LIN {X 0,Y 728.107,Z 330.531,A -85,B 0,C 180,E1 34678.19,E2 34678.19} C_VEL
LIN {X 0,Y 728.082,Z 330.529,A -85,B 0,C 180,E1 34675.632,E2 34675.632} C_VEL
LIN {X 0,Y 728.118,Z 330.525,A -85,B 0,C 180,E1 34673.04,E2 34673.04} C_VEL
LIN {X 0,Y 728.107,Z 330.532,A -85,B 0,C 180,E1 34669.995,E2 34669.995} C_VEL
LIN {X 0,Y 728.078,Z 330.53,A -85,B 0,C 180,E1 34667.503,E2 34667.503} C_VEL
LIN {X 0,Y 728.087,Z 330.528,A -85,B 0,C 180,E1 34665.043,E2 34665.043} C_VEL
LIN {X 0,Y 728.156,Z 330.532,A -85,B 0,C 180,E1 34662.12,E2 34662.12} C_VEL
LIN {X 0,Y 728.078,Z 330.532,A -85,B 0,C 180,E1 34659.406,E2 34659.406} C_VEL
LIN {X 0,Y 728.072,Z 330.53,A -85,B 0,C 180,E1 34657.021,E2 34657.021} C_VEL
LIN {X 0,Y 728.11,Z 330.528,A -85,B 0,C 180,E1 34654.44,E2 34654.44} C_VEL
LIN {X 0,Y 728.094,Z 330.533,A -85,B 0,C 180,E1 34651.416,E2 34651.416} C_VEL
LIN {X 0,Y 728.067,Z 330.532,A -85,B 0,C 180,E1 34648.977,E2 34648.977} C_VEL
LIN {X 0,Y 728.067,Z 330.527,A -85,B 0,C 180,E1 34646.615,E2 34646.615} C_VEL
LIN {X 0,Y 728.135,Z 330.531,A -85,B 0,C 180,E1 34643.93,E2 34643.93} C_VEL
LIN {X 0,Y 728.076,Z 330.534,A -85,B 0,C 180,E1 34640.993,E2 34640.993} C_VEL
LIN {X 0,Y 728.059,Z 330.532,A -85,B 0,C 180,E1 34638.594,E2 34638.594} C_VEL
LIN {X 0,Y 728.063,Z 330.531,A -85,B 0,C 180,E1 34636.256,E2 34636.256} C_VEL
LIN {X 0,Y 728.155,Z 330.51,A -85,B 0,C 180,E1 34633.433,E2 34633.433} C_VEL
LIN {X 0,Y 728.062,Z 330.521,A -85,B 0,C 180,E1 34630.589,E2 34630.589} C_VEL
LIN {X 0,Y 728.054,Z 330.543,A -85,B 0,C 180,E1 34628.235,E2 34628.235} C_VEL
LIN {X 0,Y 728.15,Z 330.769,A -85,B 0,C 180,E1 34627.473,E2 34627.473} C_VEL
LIN {X 0,Y 728.586,Z 332.326,A -85,B 0,C 180,E1 34627.328,E2 34627.328} C_VEL
LIN {X 0,Y 730.719,Z 335.448,A -85,B 0,C 180,E1 34627.132,E2 34627.132} C_VEL
LIN {X 0,Y 735.609,Z 342.898,A -85,B 0,C 180,E1 34626.692,E2 34626.692} C_VEL
LIN {X 0,Y 734.695,Z 558.029,A -85,B 0,C 180,E1 34624.049,E2 34624.049} C_VEL
LIN {X 0,Y 733.863,Z 756.602,A -85,B 0,C 180,E1 34621.662,E2 34621.662} C_VEL
LIN {X 0,Y 733.596,Z 783.313,A -85,B 0,C 180,E1 34621.191,E2 34621.191} C_VEL
LIN {X 0,Y 733.226,Z 810.458,A -85,B 0,C 180,E1 34620.549,E2 34620.549} C_VEL
LIN {X 0,Y 732.845,Z 834.995,A -85,B 0,C 180,E1 34619.817,E2 34619.817} C_VEL
LIN {X 0,Y 732.412,Z 860.75,A -85,B 0,C 180,E1 34618.903,E2 34618.903} C_VEL
LIN {X 0,Y 731.841,Z 885.617,A -85,B 0,C 180,E1 34617.854,E2 34617.854} C_VEL
LIN {X 0,Y 731.403,Z 907.627,A -85,B 0,C 180,E1 34616.789,E2 34616.789} C_VEL
LIN {X 0,Y 730.936,Z 931.895,A -85,B 0,C 180,E1 34615.458,E2 34615.458} C_VEL
LIN {X 0,Y 730.401,Z 953.79,A -85,B 0,C 180,E1 34614.085,E2 34614.085} C_VEL
LIN {X 0,Y 729.994,Z 973.19,A -85,B 0,C 180,E1 34612.732,E2 34612.732} C_VEL
LIN {X 0,Y 729.606,Z 994.463,A -85,B 0,C 180,E1 34611.077,E2 34611.077} C_VEL
LIN {X 0,Y 729.185,Z 1012.918,A -85,B 0,C 180,E1 34609.462,E2 34609.462} C_VEL
LIN {X 0,Y 728.928,Z 1030.13,A -85,B 0,C 180,E1 34607.794,E2 34607.794} C_VEL
LIN {X 0,Y 728.606,Z 1047.766,A -85,B 0,C 180,E1 34605.868,E2 34605.868} C_VEL
LIN {X 0,Y 728.411,Z 1061.269,A -85,B 0,C 180,E1 34604.214,E2 34604.214} C_VEL
LIN {X 0,Y 728.279,Z 1073.883,A -85,B 0,C 180,E1 34602.493,E2 34602.493} C_VEL
LIN {X 0,Y 728.122,Z 1087.68,A -85,B 0,C 180,E1 34600.347,E2 34600.347} C_VEL
LIN {X 0,Y 728.035,Z 1097.981,A -85,B 0,C 180,E1 34598.474,E2 34598.474} C_VEL
LIN {X 0,Y 727.947,Z 1105.598,A -85,B 0,C 180,E1 34596.888,E2 34596.888} C_VEL
LIN {X 0,Y 727.935,Z 1112.65,A -85,B 0,C 180,E1 34595.187,E2 34595.187} C_VEL
LIN {X 0,Y 727.924,Z 1118.773,A -85,B 0,C 180,E1 34593.424,E2 34593.424} C_VEL
LIN {X 0,Y 727.924,Z 1124.47,A -85,B 0,C 180,E1 34591.373,E2 34591.373} C_VEL
LIN {X 0,Y 727.915,Z 1128.569,A -85,B 0,C 180,E1 34589.276,E2 34589.276} C_VEL
LIN {X 0,Y 727.873,Z 1130.818,A -85,B 0,C 180,E1 34587.4,E2 34587.4} C_VEL
LIN {X 0,Y 727.906,Z 1131.802,A -85,B 0,C 180,E1 34585.697,E2 34585.697} C_VEL
LIN {X 0,Y 727.896,Z 1131.74,A -85,B 0,C 180,E1 34583.992,E2 34583.992} C_VEL
LIN {X 0,Y 727.916,Z 1130.33,A -85,B 0,C 180,E1 34581.94,E2 34581.94} C_VEL
LIN {X 0,Y 727.92,Z 1127.194,A -85,B 0,C 180,E1 34579.834,E2 34579.834} C_VEL
LIN {X 0,Y 727.93,Z 1122.518,A -85,B 0,C 180,E1 34577.755,E2 34577.755} C_VEL
LIN {X 0,Y 727.952,Z 1115.426,A -85,B 0,C 180,E1 34575.455,E2 34575.455} C_VEL
LIN {X 0,Y 727.985,Z 1107.016,A -85,B 0,C 180,E1 34573.341,E2 34573.341} C_VEL
LIN {X 0,Y 728.024,Z 1099.06,A -85,B 0,C 180,E1 34571.648,E2 34571.648} C_VEL
LIN {X 0,Y 728.063,Z 1089.98,A -85,B 0,C 180,E1 34569.965,E2 34569.965} C_VEL
LIN {X 0,Y 728.178,Z 1080.234,A -85,B 0,C 180,E1 34568.369,E2 34568.369} C_VEL
LIN {X 0,Y 728.35,Z 1067.162,A -85,B 0,C 180,E1 34566.464,E2 34566.464} C_VEL
LIN {X 0,Y 728.57,Z 1051.53,A -85,B 0,C 180,E1 34564.487,E2 34564.487} C_VEL
LIN {X 0,Y 728.777,Z 1037.612,A -85,B 0,C 180,E1 34562.91,E2 34562.91} C_VEL
LIN {X 0,Y 729.073,Z 1021.129,A -85,B 0,C 180,E1 34561.218,E2 34561.218} C_VEL
LIN {X 0,Y 729.412,Z 1001.74,A -85,B 0,C 180,E1 34559.45,E2 34559.45} C_VEL
LIN {X 0,Y 729.794,Z 983.502,A -85,B 0,C 180,E1 34557.959,E2 34557.959} C_VEL
LIN {X 0,Y 730.292,Z 961.036,A -85,B 0,C 180,E1 34556.31,E2 34556.31} C_VEL
LIN {X 0,Y 730.693,Z 939.861,A -85,B 0,C 180,E1 34554.936,E2 34554.936} C_VEL
LIN {X 0,Y 731.173,Z 918.904,A -85,B 0,C 180,E1 34553.719,E2 34553.719} C_VEL
LIN {X 0,Y 731.75,Z 892.704,A -85,B 0,C 180,E1 34552.383,E2 34552.383} C_VEL
LIN {X 0,Y 732.175,Z 869.485,A -85,B 0,C 180,E1 34551.36,E2 34551.36} C_VEL
LIN {X 0,Y 732.587,Z 846.861,A -85,B 0,C 180,E1 34550.494,E2 34550.494} C_VEL
LIN {X 0,Y 733.091,Z 818.282,A -85,B 0,C 180,E1 34549.578,E2 34549.578} C_VEL
LIN {X 0,Y 733.499,Z 791.667,A -85,B 0,C 180,E1 34548.898,E2 34548.898} C_VEL
LIN {X 0,Y 733.775,Z 764.714,A -85,B 0,C 180,E1 34548.375,E2 34548.375} C_VEL
LIN {X 0,Y 734.007,Z 735.424,A -85,B 0,C 180,E1 34547.977,E2 34547.977} C_VEL
LIN {X 0,Y 734.916,Z 505.975,A -85,B 0,C 180,E1 34545.23,E2 34545.23} C_VEL
LIN {X 0,Y 735.52,Z 342.703,A -85,B 0,C 180,E1 34543.209,E2 34543.209} C_VEL
LIN {X 0,Y 731.351,Z 336.17,A -85,B 0,C 180,E1 34542.832,E2 34542.832} C_VEL
LIN {X 0,Y 728.754,Z 332.691,A -85,B 0,C 180,E1 34542.601,E2 34542.601} C_VEL
LIN {X 0,Y 728.209,Z 330.851,A -85,B 0,C 180,E1 34542.459,E2 34542.459} C_VEL
LIN {X 0,Y 728.09,Z 330.538,A -85,B 0,C 180,E1 34541.753,E2 34541.753} C_VEL
LIN {X 0,Y 728.105,Z 330.514,A -85,B 0,C 180,E1 34539.165,E2 34539.165} C_VEL
LIN {X 0,Y 728.155,Z 330.527,A -85,B 0,C 180,E1 34536.189,E2 34536.189} C_VEL
LIN {X 0,Y 728.106,Z 330.53,A -85,B 0,C 180,E1 34533.379,E2 34533.379} C_VEL
LIN {X 0,Y 728.158,Z 330.533,A -85,B 0,C 180,E1 34530.554,E2 34530.554} C_VEL
LIN {X 0,Y 728.13,Z 330.526,A -85,B 0,C 180,E1 34527.618,E2 34527.618} C_VEL
LIN {X 0,Y 728.144,Z 330.534,A -85,B 0,C 180,E1 34524.778,E2 34524.778} C_VEL
LIN {X 0,Y 728.156,Z 330.527,A -85,B 0,C 180,E1 34521.734,E2 34521.734} C_VEL
LIN {X 0,Y 728.161,Z 330.717,A -85,B 0,C 180,E1 34519.286,E2 34519.286} C_VEL
LIN {X 0,Y 729.649,Z 334.269,A -85,B 0,C 180,E1 34518.869,E2 34518.869} C_VEL
LIN {X 0,Y 730.762,Z 336.329,A -85,B 0,C 180,E1 34518.633,E2 34518.633} C_VEL
LIN {X 0,Y 735.297,Z 345.332,A -85,B 0,C 180,E1 34517.648,E2 34517.648} C_VEL
LIN {X 0,Y 734.588,Z 386.425,A -85,B 0,C 180,E1 34515.111,E2 34515.111} C_VEL
LIN {X 0,Y 734.124,Z 427.552,A -85,B 0,C 180,E1 34512.689,E2 34512.689} C_VEL
LIN {X 0,Y 735.825,Z 435.852,A -85,B 0,C 180,E1 34512.457,E2 34512.457} C_VEL
LIN {X 0,Y 734.955,Z 645.516,A -85,B 0,C 180,E1 34509.852,E2 34509.852} C_VEL
LIN {X 0,Y 734.064,Z 871.192,A -85,B 0,C 180,E1 34507.146,E2 34507.146} C_VEL
LIN {X 0,Y 733.843,Z 910.622,A -85,B 0,C 180,E1 34506.646,E2 34506.646} C_VEL
LIN {X 0,Y 733.519,Z 937.557,A -85,B 0,C 180,E1 34506.146,E2 34506.146} C_VEL
LIN {X 0,Y 733.177,Z 963.48,A -85,B 0,C 180,E1 34505.511,E2 34505.511} C_VEL
LIN {X 0,Y 732.755,Z 991.376,A -85,B 0,C 180,E1 34504.654,E2 34504.654} C_VEL
LIN {X 0,Y 732.218,Z 1016.477,A -85,B 0,C 180,E1 34503.717,E2 34503.717} C_VEL
LIN {X 0,Y 731.801,Z 1037.586,A -85,B 0,C 180,E1 34502.807,E2 34502.807} C_VEL
LIN {X 0,Y 731.382,Z 1059.085,A -85,B 0,C 180,E1 34501.758,E2 34501.758} C_VEL
LIN {X 0,Y 730.853,Z 1084.154,A -85,B 0,C 180,E1 34500.365,E2 34500.365} C_VEL
LIN {X 0,Y 730.378,Z 1104.565,A -85,B 0,C 180,E1 34499.077,E2 34499.077} C_VEL
LIN {X 0,Y 730.013,Z 1122.255,A -85,B 0,C 180,E1 34497.843,E2 34497.843} C_VEL
LIN {X 0,Y 729.634,Z 1143.199,A -85,B 0,C 180,E1 34496.228,E2 34496.228} C_VEL
LIN {X 0,Y 729.209,Z 1161.707,A -85,B 0,C 180,E1 34494.617,E2 34494.617} C_VEL
LIN {X 0,Y 728.956,Z 1177.537,A -85,B 0,C 180,E1 34493.097,E2 34493.097} C_VEL
LIN {X 0,Y 728.684,Z 1194.989,A -85,B 0,C 180,E1 34491.238,E2 34491.238} C_VEL
LIN {X 0,Y 728.438,Z 1210.158,A -85,B 0,C 180,E1 34489.401,E2 34489.401} C_VEL
LIN {X 0,Y 728.264,Z 1221.836,A -85,B 0,C 180,E1 34487.828,E2 34487.828} C_VEL
LIN {X 0,Y 728.149,Z 1232.784,A -85,B 0,C 180,E1 34486.186,E2 34486.186} C_VEL
LIN {X 0,Y 728.086,Z 1244.308,A -85,B 0,C 180,E1 34484.23,E2 34484.23} C_VEL
LIN {X 0,Y 727.973,Z 1254.716,A -85,B 0,C 180,E1 34482.131,E2 34482.131} C_VEL
LIN {X 0,Y 727.956,Z 1261.878,A -85,B 0,C 180,E1 34480.431,E2 34480.431} C_VEL
LIN {X 0,Y 727.916,Z 1267.792,A -85,B 0,C 180,E1 34478.77,E2 34478.77} C_VEL
LIN {X 0,Y 727.917,Z 1273.175,A -85,B 0,C 180,E1 34476.943,E2 34476.943} C_VEL
LIN {X 0,Y 727.911,Z 1277.782,A -85,B 0,C 180,E1 34474.806,E2 34474.806} C_VEL
LIN {X 0,Y 727.912,Z 1280.541,A -85,B 0,C 180,E1 34472.756,E2 34472.756} C_VEL
LIN {X 0,Y 727.874,Z 1281.715,A -85,B 0,C 180,E1 34471.023,E2 34471.023} C_VEL
LIN {X 0,Y 727.863,Z 1281.827,A -85,B 0,C 180,E1 34469.37,E2 34469.37} C_VEL
LIN {X 0,Y 727.907,Z 1280.946,A -85,B 0,C 180,E1 34467.717,E2 34467.717} C_VEL
LIN {X 0,Y 727.919,Z 1278.803,A -85,B 0,C 180,E1 34465.825,E2 34465.825} C_VEL
LIN {X 0,Y 727.925,Z 1274.734,A -85,B 0,C 180,E1 34463.691,E2 34463.691} C_VEL
LIN {X 0,Y 727.939,Z 1269.073,A -85,B 0,C 180,E1 34461.628,E2 34461.628} C_VEL
LIN {X 0,Y 727.956,Z 1263.045,A -85,B 0,C 180,E1 34459.874,E2 34459.874} C_VEL
LIN {X 0,Y 727.966,Z 1256.145,A -85,B 0,C 180,E1 34458.191,E2 34458.191} C_VEL
LIN {X 0,Y 727.993,Z 1248.883,A -85,B 0,C 180,E1 34456.659,E2 34456.659} C_VEL
LIN {X 0,Y 728.086,Z 1240.595,A -85,B 0,C 180,E1 34455.119,E2 34455.119} C_VEL
LIN {X 0,Y 728.177,Z 1230.694,A -85,B 0,C 180,E1 34453.487,E2 34453.487} C_VEL
LIN {X 0,Y 728.347,Z 1218.342,A -85,B 0,C 180,E1 34451.677,E2 34451.677} C_VEL
LIN {X 0,Y 728.544,Z 1202.255,A -85,B 0,C 180,E1 34449.617,E2 34449.617} C_VEL
LIN {X 0,Y 728.752,Z 1188.057,A -85,B 0,C 180,E1 34448.002,E2 34448.002} C_VEL
LIN {X 0,Y 729.047,Z 1172.216,A -85,B 0,C 180,E1 34446.372,E2 34446.372} C_VEL
LIN {X 0,Y 729.421,Z 1152.324,A -85,B 0,C 180,E1 34444.548,E2 34444.548} C_VEL
LIN {X 0,Y 729.734,Z 1134.945,A -85,B 0,C 180,E1 34443.117,E2 34443.117} C_VEL
LIN {X 0,Y 730.18,Z 1115.658,A -85,B 0,C 180,E1 34441.679,E2 34441.679} C_VEL
LIN {X 0,Y 730.668,Z 1092.159,A -85,B 0,C 180,E1 34440.125,E2 34440.125} C_VEL
LIN {X 0,Y 731.057,Z 1072.423,A -85,B 0,C 180,E1 34438.961,E2 34438.961} C_VEL
LIN {X 0,Y 731.515,Z 1051.962,A -85,B 0,C 180,E1 34437.879,E2 34437.879} C_VEL
LIN {X 0,Y 732.098,Z 1026.541,A -85,B 0,C 180,E1 34436.699,E2 34436.699} C_VEL
LIN {X 0,Y 732.503,Z 1003.39,A -85,B 0,C 180,E1 34435.779,E2 34435.779} C_VEL
LIN {X 0,Y 732.865,Z 981.835,A -85,B 0,C 180,E1 34435.039,E2 34435.039} C_VEL
LIN {X 0,Y 733.236,Z 959.117,A -85,B 0,C 180,E1 34434.371,E2 34434.371} C_VEL
LIN {X 0,Y 733.615,Z 932.145,A -85,B 0,C 180,E1 34433.739,E2 34433.739} C_VEL
LIN {X 0,Y 733.88,Z 904.403,A -85,B 0,C 180,E1 34433.261,E2 34433.261} C_VEL
LIN {X 0,Y 734.857,Z 667.496,A -85,B 0,C 180,E1 34430.415,E2 34430.415} C_VEL
LIN {X 0,Y 735.696,Z 465.373,A -85,B 0,C 180,E1 34427.915,E2 34427.915} C_VEL
LIN {X 0,Y 735.645,Z 434.163,A -85,B 0,C 180,E1 34427.508,E2 34427.508} C_VEL
LIN {X 0,Y 734.005,Z 426.794,A -85,B 0,C 180,E1 34427.282,E2 34427.282} C_VEL
LIN {X 0,Y 734.649,Z 382.935,A -85,B 0,C 180,E1 34424.678,E2 34424.678} C_VEL
LIN {X 0,Y 735.253,Z 345.215,A -85,B 0,C 180,E1 34422.341,E2 34422.341} C_VEL
LIN {X 0,Y 731.832,Z 338.52,A -85,B 0,C 180,E1 34421.607,E2 34421.607} C_VEL
LIN {X 0,Y 730.082,Z 334.806,A -85,B 0,C 180,E1 34421.205,E2 34421.205} C_VEL
LIN {X 0,Y 728.288,Z 331.373,A -85,B 0,C 180,E1 34420.807,E2 34420.807} C_VEL
LIN {X 0,Y 728.146,Z 330.583,A -85,B 0,C 180,E1 34420.661,E2 34420.661} C_VEL
LIN {X 0,Y 728.135,Z 330.495,A -85,B 0,C 180,E1 34417.768,E2 34417.768} C_VEL
LIN {X 0,Y 728.138,Z 330.533,A -85,B 0,C 180,E1 34414.934,E2 34414.934} C_VEL
LIN {X 0,Y 728.155,Z 330.523,A -85,B 0,C 180,E1 34412.009,E2 34412.009} C_VEL
LIN {X 0,Y 728.154,Z 330.53,A -85,B 0,C 180,E1 34408.99,E2 34408.99} C_VEL
LIN {X 0,Y 728.15,Z 330.52,A -85,B 0,C 180,E1 34405.98,E2 34405.98} C_VEL
LIN {X 0,Y 728.159,Z 330.532,A -85,B 0,C 180,E1 34402.868,E2 34402.868} C_VEL
LIN {X 0,Y 728.138,Z 330.523,A -85,B 0,C 180,E1 34399.911,E2 34399.911} C_VEL
LIN {X 0,Y 728.15,Z 330.529,A -85,B 0,C 180,E1 34396.925,E2 34396.925} C_VEL
LIN {X 0,Y 728.122,Z 330.527,A -85,B 0,C 180,E1 34394.068,E2 34394.068} C_VEL
LIN {X 0,Y 728.154,Z 330.52,A -85,B 0,C 180,E1 34391.244,E2 34391.244} C_VEL
LIN {X 0,Y 728.139,Z 330.531,A -85,B 0,C 180,E1 34388.29,E2 34388.29} C_VEL
LIN {X 0,Y 728.141,Z 330.52,A -85,B 0,C 180,E1 34385.358,E2 34385.358} C_VEL
LIN {X 0,Y 728.153,Z 330.53,A -85,B 0,C 180,E1 34382.282,E2 34382.282} C_VEL
LIN {X 0,Y 728.119,Z 330.525,A -85,B 0,C 180,E1 34379.449,E2 34379.449} C_VEL
LIN {X 0,Y 728.151,Z 330.525,A -85,B 0,C 180,E1 34376.615,E2 34376.615} C_VEL
LIN {X 0,Y 728.12,Z 330.529,A -85,B 0,C 180,E1 34373.693,E2 34373.693} C_VEL
LIN {X 0,Y 728.14,Z 330.522,A -85,B 0,C 180,E1 34370.867,E2 34370.867} C_VEL
LIN {X 0,Y 728.142,Z 330.532,A -85,B 0,C 180,E1 34367.791,E2 34367.791} C_VEL
LIN {X 0,Y 728.156,Z 330.524,A -85,B 0,C 180,E1 34366.385,E2 34366.385} C_VEL
LIN {X 0,Y 727.165,Z 330.656,A -85,B 0,C 180,E1 34365.779,E2 34365.779} C_VEL
LIN {X 0,Y 720.764,Z 331.456,A -85,B 0,C 180,E1 34364.081,E2 34364.081} C_VEL
LIN {X 0,Y 720.198,Z 331.519,A -85,B 0,C 180,E1 34363.64,E2 34363.64} C_VEL
LIN {X 0,Y 720.172,Z 331.515,A -85,B 0,C 180,E1 34360.873,E2 34360.873} C_VEL
LIN {X 0,Y 720.217,Z 331.516,A -85,B 0,C 180,E1 34357.985,E2 34357.985} C_VEL
LIN {X 0,Y 720.173,Z 331.519,A -85,B 0,C 180,E1 34355.122,E2 34355.122} C_VEL
LIN {X 0,Y 720.188,Z 331.513,A -85,B 0,C 180,E1 34352.346,E2 34352.346} C_VEL
LIN {X 0,Y 720.198,Z 331.521,A -85,B 0,C 180,E1 34349.247,E2 34349.247} C_VEL
LIN {X 0,Y 720.162,Z 331.516,A -85,B 0,C 180,E1 34346.55,E2 34346.55} C_VEL
LIN {X 0,Y 720.219,Z 331.511,A -85,B 0,C 180,E1 34343.742,E2 34343.742} C_VEL
LIN {X 0,Y 720.171,Z 331.519,A -85,B 0,C 180,E1 34340.78,E2 34340.78} C_VEL
LIN {X 0,Y 720.16,Z 331.515,A -85,B 0,C 180,E1 34338.206,E2 34338.206} C_VEL
LIN {X 0,Y 720.221,Z 331.517,A -85,B 0,C 180,E1 34335.3,E2 34335.3} C_VEL
LIN {X 0,Y 720.161,Z 331.518,A -85,B 0,C 180,E1 34332.436,E2 34332.436} C_VEL
LIN {X 0,Y 720.161,Z 331.516,A -85,B 0,C 180,E1 34329.843,E2 34329.843} C_VEL
LIN {X 0,Y 720.223,Z 331.519,A -85,B 0,C 180,E1 34326.951,E2 34326.951} C_VEL
LIN {X 0,Y 720.153,Z 331.519,A -85,B 0,C 180,E1 34324.12,E2 34324.12} C_VEL
LIN {X 0,Y 720.158,Z 331.516,A -85,B 0,C 180,E1 34321.563,E2 34321.563} C_VEL
LIN {X 0,Y 720.221,Z 331.519,A -85,B 0,C 180,E1 34318.617,E2 34318.617} C_VEL
LIN {X 0,Y 720.147,Z 331.519,A -85,B 0,C 180,E1 34315.847,E2 34315.847} C_VEL
LIN {X 0,Y 720.153,Z 331.515,A -85,B 0,C 180,E1 34313.31,E2 34313.31} C_VEL
LIN {X 0,Y 720.22,Z 331.519,A -85,B 0,C 180,E1 34310.393,E2 34310.393} C_VEL
LIN {X 0,Y 720.143,Z 331.519,A -85,B 0,C 180,E1 34307.619,E2 34307.619} C_VEL
LIN {X 0,Y 720.143,Z 331.517,A -85,B 0,C 180,E1 34305.131,E2 34305.131} C_VEL
LIN {X 0,Y 720.223,Z 331.519,A -85,B 0,C 180,E1 34302.263,E2 34302.263} C_VEL
LIN {X 0,Y 720.14,Z 331.521,A -85,B 0,C 180,E1 34299.43,E2 34299.43} C_VEL
LIN {X 0,Y 720.134,Z 331.519,A -85,B 0,C 180,E1 34297.018,E2 34297.018} C_VEL
LIN {X 0,Y 720.168,Z 331.517,A -85,B 0,C 180,E1 34294.459,E2 34294.459} C_VEL
LIN {X 0,Y 720.157,Z 331.522,A -85,B 0,C 180,E1 34291.432,E2 34291.432} C_VEL
LIN {X 0,Y 720.128,Z 331.521,A -85,B 0,C 180,E1 34288.966,E2 34288.966} C_VEL
LIN {X 0,Y 720.131,Z 331.515,A -85,B 0,C 180,E1 34286.577,E2 34286.577} C_VEL
LIN {X 0,Y 720.219,Z 331.516,A -85,B 0,C 180,E1 34283.74,E2 34283.74} C_VEL
LIN {X 0,Y 720.131,Z 331.523,A -85,B 0,C 180,E1 34280.893,E2 34280.893} C_VEL
LIN {X 0,Y 720.121,Z 331.521,A -85,B 0,C 180,E1 34278.548,E2 34278.548} C_VEL
LIN {X 0,Y 720.128,Z 331.52,A -85,B 0,C 180,E1 34276.183,E2 34276.183} C_VEL
LIN {X 0,Y 720.207,Z 331.5,A -85,B 0,C 180,E1 34273.299,E2 34273.299} C_VEL
LIN {X 0,Y 720.12,Z 331.508,A -85,B 0,C 180,E1 34270.527,E2 34270.527} C_VEL
LIN {X 0,Y 720.115,Z 331.532,A -85,B 0,C 180,E1 34268.24,E2 34268.24} C_VEL
LIN {X 0,Y 720.148,Z 331.744,A -85,B 0,C 180,E1 34268.047,E2 34268.047} C_VEL
LIN {X 0,Y 720.558,Z 333.301,A -85,B 0,C 180,E1 34267.9,E2 34267.9} C_VEL
LIN {X 0,Y 722.666,Z 336.411,A -85,B 0,C 180,E1 34267.7,E2 34267.7} C_VEL
LIN {X 0,Y 723.885,Z 338.005,A -85,B 0,C 180,E1 34267.59,E2 34267.59} C_VEL
LIN {X 0,Y 729.608,Z 346.693,A -85,B 0,C 180,E1 34267.065,E2 34267.065} C_VEL
LIN {X 0,Y 728.452,Z 562.734,A -85,B 0,C 180,E1 34264.39,E2 34264.39} C_VEL
LIN {X 0,Y 727.429,Z 756.797,A -85,B 0,C 180,E1 34262.038,E2 34262.038} C_VEL
LIN {X 0,Y 727.091,Z 783.495,A -85,B 0,C 180,E1 34261.563,E2 34261.563} C_VEL
LIN {X 0,Y 726.621,Z 810.696,A -85,B 0,C 180,E1 34260.915,E2 34260.915} C_VEL
LIN {X 0,Y 726.143,Z 835.479,A -85,B 0,C 180,E1 34260.17,E2 34260.17} C_VEL
LIN {X 0,Y 725.597,Z 861.061,A -85,B 0,C 180,E1 34259.254,E2 34259.254} C_VEL
LIN {X 0,Y 724.916,Z 885.709,A -85,B 0,C 180,E1 34258.204,E2 34258.204} C_VEL
LIN {X 0,Y 724.343,Z 907.446,A -85,B 0,C 180,E1 34257.147,E2 34257.147} C_VEL
LIN {X 0,Y 723.75,Z 932.011,A -85,B 0,C 180,E1 34255.787,E2 34255.787} C_VEL
LIN {X 0,Y 723.094,Z 953.932,A -85,B 0,C 180,E1 34254.398,E2 34254.398} C_VEL
LIN {X 0,Y 722.552,Z 973.986,A -85,B 0,C 180,E1 34252.985,E2 34252.985} C_VEL
LIN {X 0,Y 722.007,Z 996.432,A -85,B 0,C 180,E1 34251.202,E2 34251.202} C_VEL
LIN {X 0,Y 721.525,Z 1014.133,A -85,B 0,C 180,E1 34249.625,E2 34249.625} C_VEL
LIN {X 0,Y 721.172,Z 1032.083,A -85,B 0,C 180,E1 34247.852,E2 34247.852} C_VEL
LIN {X 0,Y 720.786,Z 1048.868,A -85,B 0,C 180,E1 34245.974,E2 34245.974} C_VEL
LIN {X 0,Y 720.55,Z 1062.067,A -85,B 0,C 180,E1 34244.328,E2 34244.328} C_VEL
LIN {X 0,Y 720.359,Z 1075.904,A -85,B 0,C 180,E1 34242.402,E2 34242.402} C_VEL
LIN {X 0,Y 720.154,Z 1088.984,A -85,B 0,C 180,E1 34240.291,E2 34240.291} C_VEL
LIN {X 0,Y 720.068,Z 1098.26,A -85,B 0,C 180,E1 34238.571,E2 34238.571} C_VEL
LIN {X 0,Y 719.967,Z 1106.244,A -85,B 0,C 180,E1 34236.876,E2 34236.876} C_VEL
LIN {X 0,Y 719.946,Z 1113.054,A -85,B 0,C 180,E1 34235.196,E2 34235.196} C_VEL
LIN {X 0,Y 719.922,Z 1119.257,A -85,B 0,C 180,E1 34233.367,E2 34233.367} C_VEL
LIN {X 0,Y 719.922,Z 1124.818,A -85,B 0,C 180,E1 34231.295,E2 34231.295} C_VEL
LIN {X 0,Y 719.912,Z 1128.941,A -85,B 0,C 180,E1 34229.086,E2 34229.086} C_VEL
LIN {X 0,Y 719.863,Z 1131.019,A -85,B 0,C 180,E1 34227.193,E2 34227.193} C_VEL
LIN {X 0,Y 719.898,Z 1131.885,A -85,B 0,C 180,E1 34225.416,E2 34225.416} C_VEL
LIN {X 0,Y 719.88,Z 1131.454,A -85,B 0,C 180,E1 34223.233,E2 34223.233} C_VEL
LIN {X 0,Y 719.907,Z 1129.265,A -85,B 0,C 180,E1 34221.039,E2 34221.039} C_VEL
LIN {X 0,Y 719.911,Z 1125.392,A -85,B 0,C 180,E1 34218.882,E2 34218.882} C_VEL
LIN {X 0,Y 719.905,Z 1120.297,A -85,B 0,C 180,E1 34216.873,E2 34216.873} C_VEL
LIN {X 0,Y 719.956,Z 1113.563,A -85,B 0,C 180,E1 34214.849,E2 34214.849} C_VEL
LIN {X 0,Y 719.985,Z 1106.46,A -85,B 0,C 180,E1 34213.083,E2 34213.083} C_VEL
LIN {X 0,Y 720.07,Z 1098.432,A -85,B 0,C 180,E1 34211.372,E2 34211.372} C_VEL
LIN {X 0,Y 720.159,Z 1088.824,A -85,B 0,C 180,E1 34209.591,E2 34209.591} C_VEL
LIN {X 0,Y 720.344,Z 1075.833,A -85,B 0,C 180,E1 34207.497,E2 34207.497} C_VEL
LIN {X 0,Y 720.553,Z 1062.015,A -85,B 0,C 180,E1 34205.574,E2 34205.574} C_VEL
LIN {X 0,Y 720.792,Z 1048.542,A -85,B 0,C 180,E1 34203.898,E2 34203.898} C_VEL
LIN {X 0,Y 721.189,Z 1031.4,A -85,B 0,C 180,E1 34201.986,E2 34201.986} C_VEL
LIN {X 0,Y 721.557,Z 1013.64,A -85,B 0,C 180,E1 34200.238,E2 34200.238} C_VEL
LIN {X 0,Y 722.059,Z 994.848,A -85,B 0,C 180,E1 34198.572,E2 34198.572} C_VEL
LIN {X 0,Y 722.564,Z 973.172,A -85,B 0,C 180,E1 34196.867,E2 34196.867} C_VEL
LIN {X 0,Y 723.091,Z 954.05,A -85,B 0,C 180,E1 34195.519,E2 34195.519} C_VEL
LIN {X 0,Y 723.776,Z 930.803,A -85,B 0,C 180,E1 34194.053,E2 34194.053} C_VEL
LIN {X 0,Y 724.345,Z 907.034,A -85,B 0,C 180,E1 34192.744,E2 34192.744} C_VEL
LIN {X 0,Y 724.909,Z 885.87,A -85,B 0,C 180,E1 34191.712,E2 34191.712} C_VEL
LIN {X 0,Y 725.571,Z 861.66,A -85,B 0,C 180,E1 34190.681,E2 34190.681} C_VEL
LIN {X 0,Y 726.123,Z 836.305,A -85,B 0,C 180,E1 34189.768,E2 34189.768} C_VEL
LIN {X 0,Y 726.608,Z 811.727,A -85,B 0,C 180,E1 34189.023,E2 34189.023} C_VEL
LIN {X 0,Y 727.064,Z 784.919,A -85,B 0,C 180,E1 34188.377,E2 34188.377} C_VEL
LIN {X 0,Y 727.414,Z 758.626,A -85,B 0,C 180,E1 34187.9,E2 34187.9} C_VEL
LIN {X 0,Y 727.769,Z 701.915,A -85,B 0,C 180,E1 34187.198,E2 34187.198} C_VEL
LIN {X 0,Y 728.907,Z 476.652,A -85,B 0,C 180,E1 34184.466,E2 34184.466} C_VEL
LIN {X 0,Y 729.437,Z 346.129,A -85,B 0,C 180,E1 34182.826,E2 34182.826} C_VEL
LIN {X 0,Y 723.601,Z 337.376,A -85,B 0,C 180,E1 34182.291,E2 34182.291} C_VEL
LIN {X 0,Y 720.89,Z 333.973,A -85,B 0,C 180,E1 34182.047,E2 34182.047} C_VEL
LIN {X 0,Y 720.251,Z 332.085,A -85,B 0,C 180,E1 34181.924,E2 34181.924} C_VEL
LIN {X 0,Y 720.154,Z 331.54,A -85,B 0,C 180,E1 34181.746,E2 34181.746} C_VEL
LIN {X 0,Y 720.169,Z 331.501,A -85,B 0,C 180,E1 34179.129,E2 34179.129} C_VEL
LIN {X 0,Y 720.205,Z 331.517,A -85,B 0,C 180,E1 34176.084,E2 34176.084} C_VEL
LIN {X 0,Y 720.167,Z 331.52,A -85,B 0,C 180,E1 34173.355,E2 34173.355} C_VEL
LIN {X 0,Y 720.219,Z 331.521,A -85,B 0,C 180,E1 34170.512,E2 34170.512} C_VEL
LIN {X 0,Y 720.189,Z 331.516,A -85,B 0,C 180,E1 34167.577,E2 34167.577} C_VEL
LIN {X 0,Y 720.211,Z 331.523,A -85,B 0,C 180,E1 34164.719,E2 34164.719} C_VEL
LIN {X 0,Y 720.214,Z 331.518,A -85,B 0,C 180,E1 34161.641,E2 34161.641} C_VEL
LIN {X 0,Y 720.235,Z 331.731,A -85,B 0,C 180,E1 34159.956,E2 34159.956} C_VEL
LIN {X 0,Y 721.517,Z 334.966,A -85,B 0,C 180,E1 34159.566,E2 34159.566} C_VEL
LIN {X 0,Y 722.775,Z 337.218,A -85,B 0,C 180,E1 34159.296,E2 34159.296} C_VEL
LIN {X 0,Y 729.17,Z 349.743,A -85,B 0,C 180,E1 34157.889,E2 34157.889} C_VEL
LIN {X 0,Y 728.284,Z 390.899,A -85,B 0,C 180,E1 34155.33,E2 34155.33} C_VEL
LIN {X 0,Y 727.609,Z 426.819,A -85,B 0,C 180,E1 34153.184,E2 34153.184} C_VEL
LIN {X 0,Y 729.898,Z 437.785,A -85,B 0,C 180,E1 34152.859,E2 34152.859} C_VEL
LIN {X 0,Y 728.796,Z 647.017,A -85,B 0,C 180,E1 34150.239,E2 34150.239} C_VEL
LIN {X 0,Y 727.672,Z 872.536,A -85,B 0,C 180,E1 34147.511,E2 34147.511} C_VEL
LIN {X 0,Y 727.398,Z 911.215,A -85,B 0,C 180,E1 34147.015,E2 34147.015} C_VEL
LIN {X 0,Y 726.991,Z 938.374,A -85,B 0,C 180,E1 34146.504,E2 34146.504} C_VEL
LIN {X 0,Y 726.56,Z 964.191,A -85,B 0,C 180,E1 34145.864,E2 34145.864} C_VEL
LIN {X 0,Y 726.021,Z 991.909,A -85,B 0,C 180,E1 34145.002,E2 34145.002} C_VEL
LIN {X 0,Y 725.376,Z 1016.909,A -85,B 0,C 180,E1 34144.06,E2 34144.06} C_VEL
LIN {X 0,Y 724.836,Z 1038.081,A -85,B 0,C 180,E1 34143.139,E2 34143.139} C_VEL
LIN {X 0,Y 724.294,Z 1060.252,A -85,B 0,C 180,E1 34142.045,E2 34142.045} C_VEL
LIN {X 0,Y 723.607,Z 1085.615,A -85,B 0,C 180,E1 34140.61,E2 34140.61} C_VEL
LIN {X 0,Y 723.048,Z 1105.229,A -85,B 0,C 180,E1 34139.355,E2 34139.355} C_VEL
LIN {X 0,Y 722.551,Z 1124.265,A -85,B 0,C 180,E1 34138.007,E2 34138.007} C_VEL
LIN {X 0,Y 721.989,Z 1146.754,A -85,B 0,C 180,E1 34136.217,E2 34136.217} C_VEL
LIN {X 0,Y 721.54,Z 1163.38,A -85,B 0,C 180,E1 34134.74,E2 34134.74} C_VEL
LIN {X 0,Y 721.209,Z 1180.093,A -85,B 0,C 180,E1 34133.101,E2 34133.101} C_VEL
LIN {X 0,Y 720.833,Z 1197.834,A -85,B 0,C 180,E1 34131.14,E2 34131.14} C_VEL
LIN {X 0,Y 720.568,Z 1211.449,A -85,B 0,C 180,E1 34129.453,E2 34129.453} C_VEL
LIN {X 0,Y 720.35,Z 1223.584,A -85,B 0,C 180,E1 34127.78,E2 34127.78} C_VEL
LIN {X 0,Y 720.209,Z 1236.873,A -85,B 0,C 180,E1 34125.707,E2 34125.707} C_VEL
LIN {X 0,Y 720.048,Z 1247.243,A -85,B 0,C 180,E1 34123.818,E2 34123.818} C_VEL
LIN {X 0,Y 719.992,Z 1255.336,A -85,B 0,C 180,E1 34122.126,E2 34122.126} C_VEL
LIN {X 0,Y 719.964,Z 1262.128,A -85,B 0,C 180,E1 34120.482,E2 34120.482} C_VEL
LIN {X 0,Y 719.92,Z 1268.049,A -85,B 0,C 180,E1 34118.788,E2 34118.788} C_VEL
LIN {X 0,Y 719.919,Z 1273.37,A -85,B 0,C 180,E1 34116.94,E2 34116.94} C_VEL
LIN {X 0,Y 719.91,Z 1277.928,A -85,B 0,C 180,E1 34114.78,E2 34114.78} C_VEL
LIN {X 0,Y 719.91,Z 1280.609,A -85,B 0,C 180,E1 34112.707,E2 34112.707} C_VEL
LIN {X 0,Y 719.869,Z 1281.737,A -85,B 0,C 180,E1 34110.955,E2 34110.955} C_VEL
LIN {X 0,Y 719.863,Z 1281.827,A -85,B 0,C 180,E1 34109.363,E2 34109.363} C_VEL
LIN {X 0,Y 719.906,Z 1280.946,A -85,B 0,C 180,E1 34107.692,E2 34107.692} C_VEL
LIN {X 0,Y 719.92,Z 1278.803,A -85,B 0,C 180,E1 34105.779,E2 34105.779} C_VEL
LIN {X 0,Y 719.927,Z 1274.734,A -85,B 0,C 180,E1 34103.621,E2 34103.621} C_VEL
LIN {X 0,Y 719.944,Z 1269.073,A -85,B 0,C 180,E1 34101.534,E2 34101.534} C_VEL
LIN {X 0,Y 719.969,Z 1263.046,A -85,B 0,C 180,E1 34099.76,E2 34099.76} C_VEL
LIN {X 0,Y 719.986,Z 1256.146,A -85,B 0,C 180,E1 34098.058,E2 34098.058} C_VEL
LIN {X 0,Y 720.023,Z 1248.885,A -85,B 0,C 180,E1 34096.509,E2 34096.509} C_VEL
LIN {X 0,Y 720.136,Z 1240.597,A -85,B 0,C 180,E1 34094.951,E2 34094.951} C_VEL
LIN {X 0,Y 720.273,Z 1230.696,A -85,B 0,C 180,E1 34093.3,E2 34093.3} C_VEL
LIN {X 0,Y 720.499,Z 1217.179,A -85,B 0,C 180,E1 34091.303,E2 34091.303} C_VEL
LIN {X 0,Y 720.738,Z 1202.096,A -85,B 0,C 180,E1 34089.367,E2 34089.367} C_VEL
LIN {X 0,Y 720.993,Z 1188.059,A -85,B 0,C 180,E1 34087.753,E2 34087.753} C_VEL
LIN {X 0,Y 721.368,Z 1172.415,A -85,B 0,C 180,E1 34086.125,E2 34086.125} C_VEL
LIN {X 0,Y 721.822,Z 1152.339,A -85,B 0,C 180,E1 34084.262,E2 34084.262} C_VEL
LIN {X 0,Y 722.27,Z 1134.945,A -85,B 0,C 180,E1 34082.817,E2 34082.817} C_VEL
LIN {X 0,Y 722.804,Z 1115.595,A -85,B 0,C 180,E1 34081.359,E2 34081.359} C_VEL
LIN {X 0,Y 723.401,Z 1092.161,A -85,B 0,C 180,E1 34079.794,E2 34079.794} C_VEL
LIN {X 0,Y 723.939,Z 1072.106,A -85,B 0,C 180,E1 34078.603,E2 34078.603} C_VEL
LIN {X 0,Y 724.545,Z 1050.961,A -85,B 0,C 180,E1 34077.48,E2 34077.48} C_VEL
LIN {X 0,Y 725.223,Z 1025.426,A -85,B 0,C 180,E1 34076.294,E2 34076.294} C_VEL
LIN {X 0,Y 725.73,Z 1002.121,A -85,B 0,C 180,E1 34075.367,E2 34075.367} C_VEL
LIN {X 0,Y 726.179,Z 981.105,A -85,B 0,C 180,E1 34074.645,E2 34074.645} C_VEL
LIN {X 0,Y 726.659,Z 957.999,A -85,B 0,C 180,E1 34073.968,E2 34073.968} C_VEL
LIN {X 0,Y 727.13,Z 931.039,A -85,B 0,C 180,E1 34073.341,E2 34073.341} C_VEL
LIN {X 0,Y 727.458,Z 903.812,A -85,B 0,C 180,E1 34072.875,E2 34072.875} C_VEL
LIN {X 0,Y 728.674,Z 669.023,A -85,B 0,C 180,E1 34070.031,E2 34070.031} C_VEL
LIN {X 0,Y 729.74,Z 466.713,A -85,B 0,C 180,E1 34067.509,E2 34067.509} C_VEL
LIN {X 0,Y 729.735,Z 436.188,A -85,B 0,C 180,E1 34067.108,E2 34067.108} C_VEL
LIN {X 0,Y 727.584,Z 426.259,A -85,B 0,C 180,E1 34066.787,E2 34066.787} C_VEL
LIN {X 0,Y 728.462,Z 382.935,A -85,B 0,C 180,E1 34064.184,E2 34064.184} C_VEL
LIN {X 0,Y 729.121,Z 349.438,A -85,B 0,C 180,E1 34062.087,E2 34062.087} C_VEL
LIN {X 0,Y 724.058,Z 339.745,A -85,B 0,C 180,E1 34060.992,E2 34060.992} C_VEL
LIN {X 0,Y 721.844,Z 335.427,A -85,B 0,C 180,E1 34060.495,E2 34060.495} C_VEL
LIN {X 0,Y 720.253,Z 331.848,A -85,B 0,C 180,E1 34060.072,E2 34060.072} C_VEL
LIN {X 0,Y 720.216,Z 331.513,A -85,B 0,C 180,E1 34059.277,E2 34059.277} C_VEL
LIN {X 0,Y 720.214,Z 331.495,A -85,B 0,C 180,E1 34056.235,E2 34056.235} C_VEL
LIN {X 0,Y 720.215,Z 331.518,A -85,B 0,C 180,E1 34053.16,E2 34053.16} C_VEL
LIN {X 0,Y 720.216,Z 331.512,A -85,B 0,C 180,E1 34050.078,E2 34050.078} C_VEL
LIN {X 0,Y 720.215,Z 331.519,A -85,B 0,C 180,E1 34046.964,E2 34046.964} C_VEL
LIN {X 0,Y 720.211,Z 331.509,A -85,B 0,C 180,E1 34043.916,E2 34043.916} C_VEL
LIN {X 0,Y 720.216,Z 331.518,A -85,B 0,C 180,E1 34040.819,E2 34040.819} C_VEL
LIN {X 0,Y 720.196,Z 331.51,A -85,B 0,C 180,E1 34037.868,E2 34037.868} C_VEL
LIN {X 0,Y 720.211,Z 331.518,A -85,B 0,C 180,E1 34034.883,E2 34034.883} C_VEL
LIN {X 0,Y 720.183,Z 331.514,A -85,B 0,C 180,E1 34032.02,E2 34032.02} C_VEL
LIN {X 0,Y 720.216,Z 331.511,A -85,B 0,C 180,E1 34029.187,E2 34029.187} C_VEL
LIN {X 0,Y 720.198,Z 331.517,A -85,B 0,C 180,E1 34026.217,E2 34026.217} C_VEL
LIN {X 0,Y 720.205,Z 331.511,A -85,B 0,C 180,E1 34023.263,E2 34023.263} C_VEL
LIN {X 0,Y 720.208,Z 331.521,A -85,B 0,C 180,E1 34020.159,E2 34020.159} C_VEL
LIN {X 0,Y 720.184,Z 331.513,A -85,B 0,C 180,E1 34017.294,E2 34017.294} C_VEL
LIN {X 0,Y 720.214,Z 331.517,A -85,B 0,C 180,E1 34014.343,E2 34014.343} C_VEL
LIN {X 0,Y 720.176,Z 331.517,A -85,B 0,C 180,E1 34011.537,E2 34011.537} C_VEL
LIN {X 0,Y 720.209,Z 331.511,A -85,B 0,C 180,E1 34008.711,E2 34008.711} C_VEL
LIN {X 0,Y 720.189,Z 331.52,A -85,B 0,C 180,E1 34005.61,E2 34005.61} C_VEL
LIN {X 0,Y 720.198,Z 331.519,A -85,B 0,C 180,E1 34003.64,E2 34003.64} C_VEL
LIN {X 0,Y 719.16,Z 331.641,A -85,B 0,C 180,E1 34003.027,E2 34003.027} C_VEL
LIN {X 0,Y 712.744,Z 332.447,A -85,B 0,C 180,E1 34001.31,E2 34001.31} C_VEL
LIN {X 0,Y 712.234,Z 332.504,A -85,B 0,C 180,E1 34000.864,E2 34000.864} C_VEL
LIN {X 0,Y 712.279,Z 332.505,A -85,B 0,C 180,E1 33997.987,E2 33997.987} C_VEL
LIN {X 0,Y 712.233,Z 332.507,A -85,B 0,C 180,E1 33995.079,E2 33995.079} C_VEL
LIN {X 0,Y 712.252,Z 332.502,A -85,B 0,C 180,E1 33992.311,E2 33992.311} C_VEL
LIN {X 0,Y 712.25,Z 332.51,A -85,B 0,C 180,E1 33989.176,E2 33989.176} C_VEL
LIN {X 0,Y 712.227,Z 332.504,A -85,B 0,C 180,E1 33986.417,E2 33986.417} C_VEL
LIN {X 0,Y 712.281,Z 332.503,A -85,B 0,C 180,E1 33983.548,E2 33983.548} C_VEL
LIN {X 0,Y 712.226,Z 332.508,A -85,B 0,C 180,E1 33980.672,E2 33980.672} C_VEL
LIN {X 0,Y 712.228,Z 332.503,A -85,B 0,C 180,E1 33978.067,E2 33978.067} C_VEL
LIN {X 0,Y 712.279,Z 332.508,A -85,B 0,C 180,E1 33975.032,E2 33975.032} C_VEL
LIN {X 0,Y 712.215,Z 332.506,A -85,B 0,C 180,E1 33972.258,E2 33972.258} C_VEL
LIN {X 0,Y 712.245,Z 332.504,A -85,B 0,C 180,E1 33969.581,E2 33969.581} C_VEL
LIN {X 0,Y 712.234,Z 332.508,A -85,B 0,C 180,E1 33966.445,E2 33966.445} C_VEL
LIN {X 0,Y 712.21,Z 332.507,A -85,B 0,C 180,E1 33963.873,E2 33963.873} C_VEL
LIN {X 0,Y 712.27,Z 332.503,A -85,B 0,C 180,E1 33961.093,E2 33961.093} C_VEL
LIN {X 0,Y 712.225,Z 332.509,A -85,B 0,C 180,E1 33958.145,E2 33958.145} C_VEL
LIN {X 0,Y 712.206,Z 332.507,A -85,B 0,C 180,E1 33955.62,E2 33955.62} C_VEL
LIN {X 0,Y 712.254,Z 332.501,A -85,B 0,C 180,E1 33952.938,E2 33952.938} C_VEL
LIN {X 0,Y 712.224,Z 332.51,A -85,B 0,C 180,E1 33949.946,E2 33949.946} C_VEL
LIN {X 0,Y 712.2,Z 332.508,A -85,B 0,C 180,E1 33947.4,E2 33947.4} C_VEL
LIN {X 0,Y 712.233,Z 332.504,A -85,B 0,C 180,E1 33944.803,E2 33944.803} C_VEL
LIN {X 0,Y 712.224,Z 332.511,A -85,B 0,C 180,E1 33941.745,E2 33941.745} C_VEL
LIN {X 0,Y 712.195,Z 332.509,A -85,B 0,C 180,E1 33939.21,E2 33939.21} C_VEL
LIN {X 0,Y 712.206,Z 332.507,A -85,B 0,C 180,E1 33936.773,E2 33936.773} C_VEL
LIN {X 0,Y 712.27,Z 332.512,A -85,B 0,C 180,E1 33933.864,E2 33933.864} C_VEL
LIN {X 0,Y 712.194,Z 332.51,A -85,B 0,C 180,E1 33931.126,E2 33931.126} C_VEL
LIN {X 0,Y 712.189,Z 332.51,A -85,B 0,C 180,E1 33928.793,E2 33928.793} C_VEL
LIN {X 0,Y 712.223,Z 332.502,A -85,B 0,C 180,E1 33926.217,E2 33926.217} C_VEL
LIN {X 0,Y 712.207,Z 332.505,A -85,B 0,C 180,E1 33923.146,E2 33923.146} C_VEL
LIN {X 0,Y 712.185,Z 332.512,A -85,B 0,C 180,E1 33920.709,E2 33920.709} C_VEL
LIN {X 0,Y 712.187,Z 332.509,A -85,B 0,C 180,E1 33918.336,E2 33918.336} C_VEL
LIN {X 0,Y 712.273,Z 332.481,A -85,B 0,C 180,E1 33915.53,E2 33915.53} C_VEL
LIN {X 0,Y 712.189,Z 332.516,A -85,B 0,C 180,E1 33912.684,E2 33912.684} C_VEL
LIN {X 0,Y 712.174,Z 332.491,A -85,B 0,C 180,E1 33910.309,E2 33910.309} C_VEL
LIN {X 0,Y 712.216,Z 332.68,A -85,B 0,C 180,E1 33908.639,E2 33908.639} C_VEL
LIN {X 0,Y 712.578,Z 334.194,A -85,B 0,C 180,E1 33908.489,E2 33908.489} C_VEL
LIN {X 0,Y 714.486,Z 337.217,A -85,B 0,C 180,E1 33908.299,E2 33908.299} C_VEL
LIN {X 0,Y 715.809,Z 338.82,A -85,B 0,C 180,E1 33908.177,E2 33908.177} C_VEL
LIN {X 0,Y 718.703,Z 342.87,A -85,B 0,C 180,E1 33907.907,E2 33907.907} C_VEL
LIN {X 0,Y 723.636,Z 350.44,A -85,B 0,C 180,E1 33907.444,E2 33907.444} C_VEL
LIN {X 0,Y 722.239,Z 566.773,A -85,B 0,C 180,E1 33904.745,E2 33904.745} C_VEL
LIN {X 0,Y 721.031,Z 756.863,A -85,B 0,C 180,E1 33902.422,E2 33902.422} C_VEL
LIN {X 0,Y 720.621,Z 783.488,A -85,B 0,C 180,E1 33901.946,E2 33901.946} C_VEL
LIN {X 0,Y 720.05,Z 810.796,A -85,B 0,C 180,E1 33901.292,E2 33901.292} C_VEL
LIN {X 0,Y 719.468,Z 835.981,A -85,B 0,C 180,E1 33900.53,E2 33900.53} C_VEL
LIN {X 0,Y 718.778,Z 862.135,A -85,B 0,C 180,E1 33899.579,E2 33899.579} C_VEL
LIN {X 0,Y 718.032,Z 885.58,A -85,B 0,C 180,E1 33898.572,E2 33898.572} C_VEL
LIN {X 0,Y 717.291,Z 908.47,A -85,B 0,C 180,E1 33897.448,E2 33897.448} C_VEL
LIN {X 0,Y 716.55,Z 932.943,A -85,B 0,C 180,E1 33896.071,E2 33896.071} C_VEL
LIN {X 0,Y 715.78,Z 954.826,A -85,B 0,C 180,E1 33894.667,E2 33894.667} C_VEL
LIN {X 0,Y 715.113,Z 975.389,A -85,B 0,C 180,E1 33893.197,E2 33893.197} C_VEL
LIN {X 0,Y 714.456,Z 997.184,A -85,B 0,C 180,E1 33891.435,E2 33891.435} C_VEL
LIN {X 0,Y 713.888,Z 1014.829,A -85,B 0,C 180,E1 33889.841,E2 33889.841} C_VEL
LIN {X 0,Y 713.409,Z 1033.712,A -85,B 0,C 180,E1 33887.938,E2 33887.938} C_VEL
LIN {X 0,Y 712.975,Z 1049.619,A -85,B 0,C 180,E1 33886.125,E2 33886.125} C_VEL
LIN {X 0,Y 712.677,Z 1063.435,A -85,B 0,C 180,E1 33884.37,E2 33884.37} C_VEL
LIN {X 0,Y 712.405,Z 1078.894,A -85,B 0,C 180,E1 33882.136,E2 33882.136} C_VEL
LIN {X 0,Y 712.206,Z 1089.745,A -85,B 0,C 180,E1 33880.331,E2 33880.331} C_VEL
LIN {X 0,Y 712.1,Z 1099.152,A -85,B 0,C 180,E1 33878.547,E2 33878.547} C_VEL
LIN {X 0,Y 711.988,Z 1107.058,A -85,B 0,C 180,E1 33876.825,E2 33876.825} C_VEL
LIN {X 0,Y 711.966,Z 1115.119,A -85,B 0,C 180,E1 33874.758,E2 33874.758} C_VEL
LIN {X 0,Y 711.899,Z 1122.237,A -85,B 0,C 180,E1 33872.423,E2 33872.423} C_VEL
LIN {X 0,Y 711.913,Z 1126.863,A -85,B 0,C 180,E1 33870.373,E2 33870.373} C_VEL
LIN {X 0,Y 711.912,Z 1130.201,A -85,B 0,C 180,E1 33868.159,E2 33868.159} C_VEL
LIN {X 0,Y 711.914,Z 1131.729,A -85,B 0,C 180,E1 33865.99,E2 33865.99} C_VEL
LIN {X 0,Y 711.886,Z 1131.811,A -85,B 0,C 180,E1 33864.213,E2 33864.213} C_VEL
LIN {X 0,Y 711.878,Z 1130.821,A -85,B 0,C 180,E1 33862.452,E2 33862.452} C_VEL
LIN {X 0,Y 711.912,Z 1128.597,A -85,B 0,C 180,E1 33860.556,E2 33860.556} C_VEL
LIN {X 0,Y 711.922,Z 1124.539,A -85,B 0,C 180,E1 33858.422,E2 33858.422} C_VEL
LIN {X 0,Y 711.946,Z 1118.838,A -85,B 0,C 180,E1 33856.313,E2 33856.313} C_VEL
LIN {X 0,Y 711.943,Z 1112.915,A -85,B 0,C 180,E1 33854.56,E2 33854.56} C_VEL
LIN {X 0,Y 711.998,Z 1106.263,A -85,B 0,C 180,E1 33852.902,E2 33852.902} C_VEL
LIN {X 0,Y 712.11,Z 1098.621,A -85,B 0,C 180,E1 33851.255,E2 33851.255} C_VEL
LIN {X 0,Y 712.249,Z 1088.583,A -85,B 0,C 180,E1 33849.372,E2 33849.372} C_VEL
LIN {X 0,Y 712.467,Z 1074.895,A -85,B 0,C 180,E1 33847.16,E2 33847.16} C_VEL
LIN {X 0,Y 712.724,Z 1061.716,A -85,B 0,C 180,E1 33845.313,E2 33845.313} C_VEL
LIN {X 0,Y 713.009,Z 1048.228,A -85,B 0,C 180,E1 33843.618,E2 33843.618} C_VEL
LIN {X 0,Y 713.472,Z 1031.043,A -85,B 0,C 180,E1 33841.687,E2 33841.687} C_VEL
LIN {X 0,Y 713.955,Z 1013.251,A -85,B 0,C 180,E1 33839.92,E2 33839.92} C_VEL
LIN {X 0,Y 714.55,Z 994.426,A -85,B 0,C 180,E1 33838.236,E2 33838.236} C_VEL
LIN {X 0,Y 715.197,Z 972.672,A -85,B 0,C 180,E1 33836.513,E2 33836.513} C_VEL
LIN {X 0,Y 715.832,Z 953.504,A -85,B 0,C 180,E1 33835.152,E2 33835.152} C_VEL
LIN {X 0,Y 716.634,Z 930.172,A -85,B 0,C 180,E1 33833.672,E2 33833.672} C_VEL
LIN {X 0,Y 717.326,Z 907.048,A -85,B 0,C 180,E1 33832.39,E2 33832.39} C_VEL
LIN {X 0,Y 718.021,Z 885.849,A -85,B 0,C 180,E1 33831.35,E2 33831.35} C_VEL
LIN {X 0,Y 718.793,Z 861.591,A -85,B 0,C 180,E1 33830.31,E2 33830.31} C_VEL
LIN {X 0,Y 719.454,Z 836.192,A -85,B 0,C 180,E1 33829.389,E2 33829.389} C_VEL
LIN {X 0,Y 720.037,Z 811.705,A -85,B 0,C 180,E1 33828.642,E2 33828.642} C_VEL
LIN {X 0,Y 720.594,Z 784.795,A -85,B 0,C 180,E1 33827.992,E2 33827.992} C_VEL
LIN {X 0,Y 721.01,Z 758.411,A -85,B 0,C 180,E1 33827.511,E2 33827.511} C_VEL
LIN {X 0,Y 721.48,Z 695.381,A -85,B 0,C 180,E1 33826.729,E2 33826.729} C_VEL
LIN {X 0,Y 722.86,Z 468.99,A -85,B 0,C 180,E1 33823.956,E2 33823.956} C_VEL
LIN {X 0,Y 723.47,Z 349.996,A -85,B 0,C 180,E1 33822.448,E2 33822.448} C_VEL
LIN {X 0,Y 718.028,Z 342.109,A -85,B 0,C 180,E1 33821.943,E2 33821.943} C_VEL
LIN {X 0,Y 714.938,Z 337.598,A -85,B 0,C 180,E1 33821.651,E2 33821.651} C_VEL
LIN {X 0,Y 712.829,Z 334.75,A -85,B 0,C 180,E1 33821.452,E2 33821.452} C_VEL
LIN {X 0,Y 712.301,Z 333.038,A -85,B 0,C 180,E1 33821.334,E2 33821.334} C_VEL
LIN {X 0,Y 712.233,Z 332.511,A -85,B 0,C 180,E1 33821.12,E2 33821.12} C_VEL
LIN {X 0,Y 712.245,Z 332.51,A -85,B 0,C 180,E1 33817.986,E2 33817.986} C_VEL
LIN {X 0,Y 712.227,Z 332.512,A -85,B 0,C 180,E1 33815.269,E2 33815.269} C_VEL
LIN {X 0,Y 712.28,Z 332.508,A -85,B 0,C 180,E1 33812.347,E2 33812.347} C_VEL
LIN {X 0,Y 712.238,Z 332.507,A -85,B 0,C 180,E1 33809.456,E2 33809.456} C_VEL
LIN {X 0,Y 712.279,Z 332.511,A -85,B 0,C 180,E1 33806.613,E2 33806.613} C_VEL
LIN {X 0,Y 712.261,Z 332.506,A -85,B 0,C 180,E1 33803.55,E2 33803.55} C_VEL
LIN {X 0,Y 712.293,Z 332.647,A -85,B 0,C 180,E1 33800.617,E2 33800.617} C_VEL
LIN {X 0,Y 712.687,Z 334.23,A -85,B 0,C 180,E1 33800.435,E2 33800.435} C_VEL
LIN {X 0,Y 714.926,Z 338.303,A -85,B 0,C 180,E1 33799.957,E2 33799.957} C_VEL
LIN {X 0,Y 722.086,Z 352.311,A -85,B 0,C 180,E1 33798.343,E2 33798.343} C_VEL
LIN {X 0,Y 723.049,Z 354.396,A -85,B 0,C 180,E1 33798.119,E2 33798.119} C_VEL
LIN {X 0,Y 721.97,Z 396.267,A -85,B 0,C 180,E1 33795.499,E2 33795.499} C_VEL
LIN {X 0,Y 721.343,Z 427.437,A -85,B 0,C 180,E1 33793.635,E2 33793.635} C_VEL
LIN {X 0,Y 724.008,Z 439.747,A -85,B 0,C 180,E1 33793.267,E2 33793.267} C_VEL
LIN {X 0,Y 722.67,Z 648.544,A -85,B 0,C 180,E1 33790.632,E2 33790.632} C_VEL
LIN {X 0,Y 721.309,Z 874.139,A -85,B 0,C 180,E1 33787.881,E2 33787.881} C_VEL
LIN {X 0,Y 720.983,Z 911.849,A -85,B 0,C 180,E1 33787.391,E2 33787.391} C_VEL
LIN {X 0,Y 720.488,Z 939.156,A -85,B 0,C 180,E1 33786.87,E2 33786.87} C_VEL
LIN {X 0,Y 719.974,Z 964.761,A -85,B 0,C 180,E1 33786.227,E2 33786.227} C_VEL
LIN {X 0,Y 719.335,Z 991.904,A -85,B 0,C 180,E1 33785.376,E2 33785.376} C_VEL
LIN {X 0,Y 718.599,Z 1016.484,A -85,B 0,C 180,E1 33784.445,E2 33784.445} C_VEL
LIN {X 0,Y 717.941,Z 1037.692,A -85,B 0,C 180,E1 33783.518,E2 33783.518} C_VEL
LIN {X 0,Y 717.252,Z 1059.982,A -85,B 0,C 180,E1 33782.412,E2 33782.412} C_VEL
LIN {X 0,Y 716.464,Z 1084.883,A -85,B 0,C 180,E1 33780.995,E2 33780.995} C_VEL
LIN {X 0,Y 715.788,Z 1104.569,A -85,B 0,C 180,E1 33779.729,E2 33779.729} C_VEL
LIN {X 0,Y 715.193,Z 1122.806,A -85,B 0,C 180,E1 33778.431,E2 33778.431} C_VEL
LIN {X 0,Y 714.536,Z 1144.214,A -85,B 0,C 180,E1 33776.736,E2 33776.736} C_VEL
LIN {X 0,Y 713.97,Z 1162.449,A -85,B 0,C 180,E1 33775.108,E2 33775.108} C_VEL
LIN {X 0,Y 713.521,Z 1178.393,A -85,B 0,C 180,E1 33773.539,E2 33773.539} C_VEL
LIN {X 0,Y 713.06,Z 1197.125,A -85,B 0,C 180,E1 33771.468,E2 33771.468} C_VEL
LIN {X 0,Y 712.725,Z 1211.123,A -85,B 0,C 180,E1 33769.719,E2 33769.719} C_VEL
LIN {X 0,Y 712.48,Z 1223.004,A -85,B 0,C 180,E1 33768.068,E2 33768.068} C_VEL
LIN {X 0,Y 712.274,Z 1235.899,A -85,B 0,C 180,E1 33766.054,E2 33766.054} C_VEL
LIN {X 0,Y 712.103,Z 1247.244,A -85,B 0,C 180,E1 33763.976,E2 33763.976} C_VEL
LIN {X 0,Y 712.021,Z 1255.433,A -85,B 0,C 180,E1 33762.242,E2 33762.242} C_VEL
LIN {X 0,Y 711.975,Z 1262.435,A -85,B 0,C 180,E1 33760.519,E2 33760.519} C_VEL
LIN {X 0,Y 711.924,Z 1268.306,A -85,B 0,C 180,E1 33758.806,E2 33758.806} C_VEL
LIN {X 0,Y 711.921,Z 1273.566,A -85,B 0,C 180,E1 33756.937,E2 33756.937} C_VEL
LIN {X 0,Y 711.913,Z 1277.928,A -85,B 0,C 180,E1 33754.834,E2 33754.834} C_VEL
LIN {X 0,Y 711.911,Z 1280.609,A -85,B 0,C 180,E1 33752.737,E2 33752.737} C_VEL
LIN {X 0,Y 711.871,Z 1281.737,A -85,B 0,C 180,E1 33750.966,E2 33750.966} C_VEL
LIN {X 0,Y 711.863,Z 1281.827,A -85,B 0,C 180,E1 33749.356,E2 33749.356} C_VEL
LIN {X 0,Y 711.905,Z 1280.946,A -85,B 0,C 180,E1 33747.666,E2 33747.666} C_VEL
LIN {X 0,Y 711.92,Z 1278.803,A -85,B 0,C 180,E1 33745.731,E2 33745.731} C_VEL
LIN {X 0,Y 711.928,Z 1274.734,A -85,B 0,C 180,E1 33743.549,E2 33743.549} C_VEL
LIN {X 0,Y 711.947,Z 1269.074,A -85,B 0,C 180,E1 33741.439,E2 33741.439} C_VEL
LIN {X 0,Y 711.98,Z 1263.047,A -85,B 0,C 180,E1 33739.644,E2 33739.644} C_VEL
LIN {X 0,Y 712.008,Z 1256.147,A -85,B 0,C 180,E1 33737.922,E2 33737.922} C_VEL
LIN {X 0,Y 712.061,Z 1248.825,A -85,B 0,C 180,E1 33736.343,E2 33736.343} C_VEL
LIN {X 0,Y 712.195,Z 1240.599,A -85,B 0,C 180,E1 33734.779,E2 33734.779} C_VEL
LIN {X 0,Y 712.371,Z 1230.698,A -85,B 0,C 180,E1 33733.11,E2 33733.11} C_VEL
LIN {X 0,Y 712.639,Z 1217.181,A -85,B 0,C 180,E1 33731.089,E2 33731.089} C_VEL
LIN {X 0,Y 712.945,Z 1201.641,A -85,B 0,C 180,E1 33729.076,E2 33729.076} C_VEL
LIN {X 0,Y 713.255,Z 1188.014,A -85,B 0,C 180,E1 33727.494,E2 33727.494} C_VEL
LIN {X 0,Y 713.712,Z 1172.417,A -85,B 0,C 180,E1 33725.853,E2 33725.853} C_VEL
LIN {X 0,Y 714.249,Z 1152.636,A -85,B 0,C 180,E1 33723.994,E2 33723.994} C_VEL
LIN {X 0,Y 714.801,Z 1135.499,A -85,B 0,C 180,E1 33722.554,E2 33722.554} C_VEL
LIN {X 0,Y 715.403,Z 1116.81,A -85,B 0,C 180,E1 33721.126,E2 33721.126} C_VEL
LIN {X 0,Y 716.163,Z 1092.529,A -85,B 0,C 180,E1 33719.479,E2 33719.479} C_VEL
LIN {X 0,Y 716.84,Z 1072.428,A -85,B 0,C 180,E1 33718.274,E2 33718.274} C_VEL
LIN {X 0,Y 717.527,Z 1051.903,A -85,B 0,C 180,E1 33717.172,E2 33717.172} C_VEL
LIN {X 0,Y 718.347,Z 1026.548,A -85,B 0,C 180,E1 33715.975,E2 33715.975} C_VEL
LIN {X 0,Y 718.978,Z 1002.227,A -85,B 0,C 180,E1 33714.998,E2 33714.998} C_VEL
LIN {X 0,Y 719.537,Z 980.471,A -85,B 0,C 180,E1 33714.247,E2 33714.247} C_VEL
LIN {X 0,Y 720.134,Z 957.209,A -85,B 0,C 180,E1 33713.568,E2 33713.568} C_VEL
LIN {X 0,Y 720.673,Z 930.235,A -85,B 0,C 180,E1 33712.942,E2 33712.942} C_VEL
LIN {X 0,Y 721.072,Z 903.24,A -85,B 0,C 180,E1 33712.482,E2 33712.482} C_VEL
LIN {X 0,Y 722.527,Z 670.041,A -85,B 0,C 180,E1 33709.634,E2 33709.634} C_VEL
LIN {X 0,Y 723.823,Z 467.731,A -85,B 0,C 180,E1 33707.092,E2 33707.092} C_VEL
LIN {X 0,Y 723.857,Z 438.257,A -85,B 0,C 180,E1 33706.702,E2 33706.702} C_VEL
LIN {X 0,Y 721.254,Z 426.813,A -85,B 0,C 180,E1 33706.34,E2 33706.34} C_VEL
LIN {X 0,Y 722.281,Z 384.338,A -85,B 0,C 180,E1 33703.767,E2 33703.767} C_VEL
LIN {X 0,Y 723.024,Z 354.054,A -85,B 0,C 180,E1 33701.856,E2 33701.856} C_VEL
LIN {X 0,Y 716.179,Z 340.795,A -85,B 0,C 180,E1 33700.334,E2 33700.334} C_VEL
LIN {X 0,Y 714.254,Z 336.874,A -85,B 0,C 180,E1 33699.878,E2 33699.878} C_VEL
LIN {X 0,Y 712.7,Z 334.285,A -85,B 0,C 180,E1 33699.565,E2 33699.565} C_VEL
LIN {X 0,Y 712.289,Z 332.612,A -85,B 0,C 180,E1 33699.355,E2 33699.355} C_VEL
LIN {X 0,Y 712.27,Z 332.473,A -85,B 0,C 180,E1 33696.315,E2 33696.315} C_VEL
LIN {X 0,Y 712.276,Z 332.505,A -85,B 0,C 180,E1 33693.212,E2 33693.212} C_VEL
LIN {X 0,Y 712.272,Z 332.502,A -85,B 0,C 180,E1 33690.148,E2 33690.148} C_VEL
LIN {X 0,Y 712.279,Z 332.508,A -85,B 0,C 180,E1 33687.054,E2 33687.054} C_VEL
LIN {X 0,Y 712.262,Z 332.499,A -85,B 0,C 180,E1 33684.023,E2 33684.023} C_VEL
LIN {X 0,Y 712.277,Z 332.506,A -85,B 0,C 180,E1 33680.976,E2 33680.976} C_VEL
LIN {X 0,Y 712.248,Z 332.501,A -85,B 0,C 180,E1 33678.074,E2 33678.074} C_VEL
LIN {X 0,Y 712.269,Z 332.502,A -85,B 0,C 180,E1 33675.219,E2 33675.219} C_VEL
LIN {X 0,Y 712.254,Z 332.505,A -85,B 0,C 180,E1 33672.297,E2 33672.297} C_VEL
LIN {X 0,Y 712.275,Z 332.499,A -85,B 0,C 180,E1 33669.372,E2 33669.372} C_VEL
LIN {X 0,Y 712.265,Z 332.507,A -85,B 0,C 180,E1 33666.286,E2 33666.286} C_VEL
LIN {X 0,Y 712.262,Z 332.501,A -85,B 0,C 180,E1 33663.3,E2 33663.3} C_VEL
LIN {X 0,Y 712.27,Z 332.51,A -85,B 0,C 180,E1 33660.161,E2 33660.161} C_VEL
LIN {X 0,Y 712.248,Z 332.502,A -85,B 0,C 180,E1 33657.264,E2 33657.264} C_VEL
LIN {X 0,Y 712.277,Z 332.508,A -85,B 0,C 180,E1 33654.28,E2 33654.28} C_VEL
LIN {X 0,Y 712.234,Z 332.506,A -85,B 0,C 180,E1 33651.442,E2 33651.442} C_VEL
LIN {X 0,Y 712.279,Z 332.5,A -85,B 0,C 180,E1 33648.584,E2 33648.584} C_VEL
LIN {X 0,Y 712.251,Z 332.509,A -85,B 0,C 180,E1 33645.612,E2 33645.612} C_VEL
LIN {X 0,Y 712.244,Z 332.5,A -85,B 0,C 180,E1 33642.77,E2 33642.77} C_VEL
LIN {X 0,Y 712.234,Z 332.504,A -85,B 0,C 180,E1 33640.864,E2 33640.864} C_VEL
LIN {X 0,Y 711.274,Z 332.627,A -85,B 0,C 180,E1 33640.245,E2 33640.245} C_VEL
LIN {X 0,Y 704.875,Z 333.423,A -85,B 0,C 180,E1 33638.509,E2 33638.509} C_VEL
LIN {X 0,Y 704.341,Z 333.492,A -85,B 0,C 180,E1 33638.057,E2 33638.057} C_VEL
LIN {X 0,Y 704.296,Z 333.497,A -85,B 0,C 180,E1 33635.118,E2 33635.118} C_VEL
LIN {X 0,Y 704.31,Z 333.491,A -85,B 0,C 180,E1 33632.339,E2 33632.339} C_VEL
LIN {X 0,Y 704.311,Z 333.499,A -85,B 0,C 180,E1 33629.169,E2 33629.169} C_VEL
LIN {X 0,Y 704.288,Z 333.494,A -85,B 0,C 180,E1 33626.446,E2 33626.446} C_VEL
LIN {X 0,Y 704.342,Z 333.493,A -85,B 0,C 180,E1 33623.5,E2 33623.5} C_VEL
LIN {X 0,Y 704.285,Z 333.496,A -85,B 0,C 180,E1 33620.608,E2 33620.608} C_VEL
LIN {X 0,Y 704.3,Z 333.491,A -85,B 0,C 180,E1 33617.925,E2 33617.925} C_VEL
LIN {X 0,Y 704.307,Z 333.498,A -85,B 0,C 180,E1 33614.761,E2 33614.761} C_VEL
LIN {X 0,Y 704.278,Z 333.493,A -85,B 0,C 180,E1 33612.053,E2 33612.053} C_VEL
LIN {X 0,Y 704.346,Z 333.494,A -85,B 0,C 180,E1 33609.177,E2 33609.177} C_VEL
LIN {X 0,Y 704.28,Z 333.496,A -85,B 0,C 180,E1 33606.253,E2 33606.253} C_VEL
LIN {X 0,Y 704.282,Z 333.495,A -85,B 0,C 180,E1 33603.62,E2 33603.62} C_VEL
LIN {X 0,Y 704.343,Z 333.499,A -85,B 0,C 180,E1 33600.639,E2 33600.639} C_VEL
LIN {X 0,Y 704.268,Z 333.497,A -85,B 0,C 180,E1 33597.846,E2 33597.846} C_VEL
LIN {X 0,Y 704.287,Z 333.494,A -85,B 0,C 180,E1 33595.262,E2 33595.262} C_VEL
LIN {X 0,Y 704.307,Z 333.499,A -85,B 0,C 180,E1 33592.187,E2 33592.187} C_VEL
LIN {X 0,Y 704.264,Z 333.498,A -85,B 0,C 180,E1 33589.576,E2 33589.576} C_VEL
LIN {X 0,Y 704.281,Z 333.495,A -85,B 0,C 180,E1 33587.005,E2 33587.005} C_VEL
LIN {X 0,Y 704.296,Z 333.5,A -85,B 0,C 180,E1 33583.882,E2 33583.882} C_VEL
LIN {X 0,Y 704.259,Z 333.499,A -85,B 0,C 180,E1 33581.299,E2 33581.299} C_VEL
LIN {X 0,Y 704.276,Z 333.497,A -85,B 0,C 180,E1 33578.738,E2 33578.738} C_VEL
LIN {X 0,Y 704.289,Z 333.498,A -85,B 0,C 180,E1 33575.622,E2 33575.622} C_VEL
LIN {X 0,Y 704.254,Z 333.498,A -85,B 0,C 180,E1 33573.093,E2 33573.093} C_VEL
LIN {X 0,Y 704.259,Z 333.498,A -85,B 0,C 180,E1 33570.651,E2 33570.651} C_VEL
LIN {X 0,Y 704.333,Z 333.489,A -85,B 0,C 180,E1 33567.722,E2 33567.722} C_VEL
LIN {X 0,Y 704.253,Z 333.501,A -85,B 0,C 180,E1 33564.95,E2 33564.95} C_VEL
LIN {X 0,Y 704.246,Z 333.493,A -85,B 0,C 180,E1 33562.577,E2 33562.577} C_VEL
LIN {X 0,Y 704.281,Z 333.5,A -85,B 0,C 180,E1 33560.026,E2 33560.026} C_VEL
LIN {X 0,Y 704.265,Z 333.499,A -85,B 0,C 180,E1 33556.954,E2 33556.954} C_VEL
LIN {X 0,Y 704.237,Z 333.462,A -85,B 0,C 180,E1 33554.519,E2 33554.519} C_VEL
LIN {X 0,Y 704.244,Z 333.507,A -85,B 0,C 180,E1 33552.141,E2 33552.141} C_VEL
LIN {X 0,Y 704.348,Z 333.588,A -85,B 0,C 180,E1 33549.251,E2 33549.251} C_VEL
LIN {X 0,Y 704.664,Z 335.026,A -85,B 0,C 180,E1 33549.092,E2 33549.092} C_VEL
LIN {X 0,Y 706.6,Z 338.192,A -85,B 0,C 180,E1 33548.892,E2 33548.892} C_VEL
LIN {X 0,Y 707.889,Z 339.792,A -85,B 0,C 180,E1 33548.769,E2 33548.769} C_VEL
LIN {X 0,Y 710.674,Z 343.792,A -85,B 0,C 180,E1 33548.5,E2 33548.5} C_VEL
LIN {X 0,Y 717.697,Z 354.069,A -85,B 0,C 180,E1 33547.832,E2 33547.832} C_VEL
LIN {X 0,Y 716.056,Z 570.643,A -85,B 0,C 180,E1 33545.109,E2 33545.109} C_VEL
LIN {X 0,Y 714.668,Z 756.854,A -85,B 0,C 180,E1 33542.815,E2 33542.815} C_VEL
LIN {X 0,Y 714.183,Z 783.486,A -85,B 0,C 180,E1 33542.336,E2 33542.336} C_VEL
LIN {X 0,Y 713.521,Z 810.77,A -85,B 0,C 180,E1 33541.679,E2 33541.679} C_VEL
LIN {X 0,Y 712.829,Z 835.954,A -85,B 0,C 180,E1 33540.914,E2 33540.914} C_VEL
LIN {X 0,Y 712.033,Z 862.033,A -85,B 0,C 180,E1 33539.959,E2 33539.959} C_VEL
LIN {X 0,Y 711.17,Z 885.661,A -85,B 0,C 180,E1 33538.937,E2 33538.937} C_VEL
LIN {X 0,Y 710.338,Z 907.577,A -85,B 0,C 180,E1 33537.854,E2 33537.854} C_VEL
LIN {X 0,Y 709.435,Z 932.275,A -85,B 0,C 180,E1 33536.463,E2 33536.463} C_VEL
LIN {X 0,Y 708.547,Z 954.214,A -85,B 0,C 180,E1 33535.045,E2 33535.045} C_VEL
LIN {X 0,Y 707.783,Z 974.214,A -85,B 0,C 180,E1 33533.607,E2 33533.607} C_VEL
LIN {X 0,Y 706.976,Z 996.192,A -85,B 0,C 180,E1 33531.826,E2 33531.826} C_VEL
LIN {X 0,Y 706.331,Z 1013.858,A -85,B 0,C 180,E1 33530.22,E2 33530.22} C_VEL
LIN {X 0,Y 705.733,Z 1032.301,A -85,B 0,C 180,E1 33528.358,E2 33528.358} C_VEL
LIN {X 0,Y 705.21,Z 1049.017,A -85,B 0,C 180,E1 33526.444,E2 33526.444} C_VEL
LIN {X 0,Y 704.858,Z 1063.031,A -85,B 0,C 180,E1 33524.649,E2 33524.649} C_VEL
LIN {X 0,Y 704.518,Z 1078.26,A -85,B 0,C 180,E1 33522.439,E2 33522.439} C_VEL
LIN {X 0,Y 704.276,Z 1090.067,A -85,B 0,C 180,E1 33520.45,E2 33520.45} C_VEL
LIN {X 0,Y 704.134,Z 1099.432,A -85,B 0,C 180,E1 33518.648,E2 33518.648} C_VEL
LIN {X 0,Y 704.013,Z 1108.086,A -85,B 0,C 180,E1 33516.722,E2 33516.722} C_VEL
LIN {X 0,Y 703.963,Z 1116.684,A -85,B 0,C 180,E1 33514.389,E2 33514.389} C_VEL
LIN {X 0,Y 703.922,Z 1123.052,A -85,B 0,C 180,E1 33512.186,E2 33512.186} C_VEL
LIN {X 0,Y 703.92,Z 1127.819,A -85,B 0,C 180,E1 33509.906,E2 33509.906} C_VEL
LIN {X 0,Y 703.909,Z 1130.6,A -85,B 0,C 180,E1 33507.755,E2 33507.755} C_VEL
LIN {X 0,Y 703.912,Z 1131.771,A -85,B 0,C 180,E1 33505.855,E2 33505.855} C_VEL
LIN {X 0,Y 703.891,Z 1131.773,A -85,B 0,C 180,E1 33504.06,E2 33504.06} C_VEL
LIN {X 0,Y 703.918,Z 1130.493,A -85,B 0,C 180,E1 33502.025,E2 33502.025} C_VEL
LIN {X 0,Y 703.921,Z 1127.622,A -85,B 0,C 180,E1 33499.893,E2 33499.893} C_VEL
LIN {X 0,Y 703.937,Z 1122.982,A -85,B 0,C 180,E1 33497.696,E2 33497.696} C_VEL
LIN {X 0,Y 703.963,Z 1116.844,A -85,B 0,C 180,E1 33495.572,E2 33495.572} C_VEL
LIN {X 0,Y 704.041,Z 1108.571,A -85,B 0,C 180,E1 33493.302,E2 33493.302} C_VEL
LIN {X 0,Y 704.137,Z 1099.626,A -85,B 0,C 180,E1 33491.301,E2 33491.301} C_VEL
LIN {X 0,Y 704.288,Z 1089.716,A -85,B 0,C 180,E1 33489.397,E2 33489.397} C_VEL
LIN {X 0,Y 704.51,Z 1077.938,A -85,B 0,C 180,E1 33487.421,E2 33487.421} C_VEL
LIN {X 0,Y 704.85,Z 1063.262,A -85,B 0,C 180,E1 33485.291,E2 33485.291} C_VEL
LIN {X 0,Y 705.206,Z 1049.068,A -85,B 0,C 180,E1 33483.473,E2 33483.473} C_VEL
LIN {X 0,Y 705.74,Z 1032.235,A -85,B 0,C 180,E1 33481.543,E2 33481.543} C_VEL
LIN {X 0,Y 706.344,Z 1013.718,A -85,B 0,C 180,E1 33479.676,E2 33479.676} C_VEL
LIN {X 0,Y 707.028,Z 994.942,A -85,B 0,C 180,E1 33477.974,E2 33477.974} C_VEL
LIN {X 0,Y 707.813,Z 973.258,A -85,B 0,C 180,E1 33476.234,E2 33476.234} C_VEL
LIN {X 0,Y 708.577,Z 953.549,A -85,B 0,C 180,E1 33474.818,E2 33474.818} C_VEL
LIN {X 0,Y 709.498,Z 930.206,A -85,B 0,C 180,E1 33473.323,E2 33473.323} C_VEL
LIN {X 0,Y 710.347,Z 907.053,A -85,B 0,C 180,E1 33472.03,E2 33472.03} C_VEL
LIN {X 0,Y 711.162,Z 885.828,A -85,B 0,C 180,E1 33470.981,E2 33470.981} C_VEL
LIN {X 0,Y 712.012,Z 862.531,A -85,B 0,C 180,E1 33469.972,E2 33469.972} C_VEL
LIN {X 0,Y 712.815,Z 836.081,A -85,B 0,C 180,E1 33469.002,E2 33469.002} C_VEL
LIN {X 0,Y 713.508,Z 811.497,A -85,B 0,C 180,E1 33468.25,E2 33468.25} C_VEL
LIN {X 0,Y 714.163,Z 784.311,A -85,B 0,C 180,E1 33467.592,E2 33467.592} C_VEL
LIN {X 0,Y 714.649,Z 757.849,A -85,B 0,C 180,E1 33467.11,E2 33467.11} C_VEL
LIN {X 0,Y 715.318,Z 676.208,A -85,B 0,C 180,E1 33466.097,E2 33466.097} C_VEL
LIN {X 0,Y 716.951,Z 450.714,A -85,B 0,C 180,E1 33463.305,E2 33463.305} C_VEL
LIN {X 0,Y 717.602,Z 353.591,A -85,B 0,C 180,E1 33462.065,E2 33462.065} C_VEL
LIN {X 0,Y 710.124,Z 343.166,A -85,B 0,C 180,E1 33461.36,E2 33461.36} C_VEL
LIN {X 0,Y 706.974,Z 338.52,A -85,B 0,C 180,E1 33461.052,E2 33461.052} C_VEL
LIN {X 0,Y 704.835,Z 335.453,A -85,B 0,C 180,E1 33460.84,E2 33460.84} C_VEL
LIN {X 0,Y 704.412,Z 333.938,A -85,B 0,C 180,E1 33460.722,E2 33460.722} C_VEL
LIN {X 0,Y 704.342,Z 333.465,A -85,B 0,C 180,E1 33460.494,E2 33460.494} C_VEL
LIN {X 0,Y 704.284,Z 333.502,A -85,B 0,C 180,E1 33457.636,E2 33457.636} C_VEL
LIN {X 0,Y 704.32,Z 333.502,A -85,B 0,C 180,E1 33454.882,E2 33454.882} C_VEL
LIN {X 0,Y 704.312,Z 333.495,A -85,B 0,C 180,E1 33451.787,E2 33451.787} C_VEL
LIN {X 0,Y 704.311,Z 333.501,A -85,B 0,C 180,E1 33448.98,E2 33448.98} C_VEL
LIN {X 0,Y 704.344,Z 333.493,A -85,B 0,C 180,E1 33445.893,E2 33445.893} C_VEL
LIN {X 0,Y 704.318,Z 333.501,A -85,B 0,C 180,E1 33442.889,E2 33442.889} C_VEL
LIN {X 0,Y 704.354,Z 333.767,A -85,B 0,C 180,E1 33440.97,E2 33440.97} C_VEL
LIN {X 0,Y 706.44,Z 339.061,A -85,B 0,C 180,E1 33440.542,E2 33440.542} C_VEL
LIN {X 0,Y 709.317,Z 343.73,A -85,B 0,C 180,E1 33440.104,E2 33440.104} C_VEL
LIN {X 0,Y 716.487,Z 357.767,A -85,B 0,C 180,E1 33438.48,E2 33438.48} C_VEL
LIN {X 0,Y 716.936,Z 359.075,A -85,B 0,C 180,E1 33438.351,E2 33438.351} C_VEL
LIN {X 0,Y 715.663,Z 401.635,A -85,B 0,C 180,E1 33435.67,E2 33435.67} C_VEL
LIN {X 0,Y 714.944,Z 426.793,A -85,B 0,C 180,E1 33434.144,E2 33434.144} C_VEL
LIN {X 0,Y 718.155,Z 441.781,A -85,B 0,C 180,E1 33433.68,E2 33433.68} C_VEL
LIN {X 0,Y 716.577,Z 650.071,A -85,B 0,C 180,E1 33431.031,E2 33431.031} C_VEL
LIN {X 0,Y 714.979,Z 875.285,A -85,B 0,C 180,E1 33428.262,E2 33428.262} C_VEL
LIN {X 0,Y 714.599,Z 912.245,A -85,B 0,C 180,E1 33427.776,E2 33427.776} C_VEL
LIN {X 0,Y 714.023,Z 939.566,A -85,B 0,C 180,E1 33427.249,E2 33427.249} C_VEL
LIN {X 0,Y 713.43,Z 964.743,A -85,B 0,C 180,E1 33426.613,E2 33426.613} C_VEL
LIN {X 0,Y 712.681,Z 991.901,A -85,B 0,C 180,E1 33425.756,E2 33425.756} C_VEL
LIN {X 0,Y 711.838,Z 1016.488,A -85,B 0,C 180,E1 33424.819,E2 33424.819} C_VEL
LIN {X 0,Y 711.071,Z 1037.695,A -85,B 0,C 180,E1 33423.886,E2 33423.886} C_VEL
LIN {X 0,Y 710.259,Z 1059.22,A -85,B 0,C 180,E1 33422.812,E2 33422.812} C_VEL
LIN {X 0,Y 709.314,Z 1084.88,A -85,B 0,C 180,E1 33421.343,E2 33421.343} C_VEL
LIN {X 0,Y 708.53,Z 1104.57,A -85,B 0,C 180,E1 33420.064,E2 33420.064} C_VEL
LIN {X 0,Y 707.823,Z 1122.863,A -85,B 0,C 180,E1 33418.75,E2 33418.75} C_VEL
LIN {X 0,Y 707.03,Z 1144.215,A -85,B 0,C 180,E1 33417.043,E2 33417.043} C_VEL
LIN {X 0,Y 706.386,Z 1162.45,A -85,B 0,C 180,E1 33415.397,E2 33415.397} C_VEL
LIN {X 0,Y 705.83,Z 1178.75,A -85,B 0,C 180,E1 33413.775,E2 33413.775} C_VEL
LIN {X 0,Y 705.286,Z 1197.127,A -85,B 0,C 180,E1 33411.717,E2 33411.717} C_VEL
LIN {X 0,Y 704.891,Z 1210.809,A -85,B 0,C 180,E1 33409.99,E2 33409.99} C_VEL
LIN {X 0,Y 704.615,Z 1223.006,A -85,B 0,C 180,E1 33408.277,E2 33408.277} C_VEL
LIN {X 0,Y 704.341,Z 1236.406,A -85,B 0,C 180,E1 33406.155,E2 33406.155} C_VEL
LIN {X 0,Y 704.156,Z 1247.403,A -85,B 0,C 180,E1 33404.104,E2 33404.104} C_VEL
LIN {X 0,Y 704.057,Z 1255.434,A -85,B 0,C 180,E1 33402.383,E2 33402.383} C_VEL
LIN {X 0,Y 703.982,Z 1262.436,A -85,B 0,C 180,E1 33400.64,E2 33400.64} C_VEL
LIN {X 0,Y 703.916,Z 1268.051,A -85,B 0,C 180,E1 33398.989,E2 33398.989} C_VEL
LIN {X 0,Y 703.934,Z 1273.37,A -85,B 0,C 180,E1 33397.098,E2 33397.098} C_VEL
LIN {X 0,Y 703.917,Z 1277.928,A -85,B 0,C 180,E1 33394.889,E2 33394.889} C_VEL
LIN {X 0,Y 703.912,Z 1280.609,A -85,B 0,C 180,E1 33392.768,E2 33392.768} C_VEL
LIN {X 0,Y 703.871,Z 1281.737,A -85,B 0,C 180,E1 33390.977,E2 33390.977} C_VEL
LIN {X 0,Y 703.863,Z 1281.827,A -85,B 0,C 180,E1 33389.349,E2 33389.349} C_VEL
LIN {X 0,Y 703.905,Z 1280.946,A -85,B 0,C 180,E1 33387.639,E2 33387.639} C_VEL
LIN {X 0,Y 703.918,Z 1278.803,A -85,B 0,C 180,E1 33385.682,E2 33385.682} C_VEL
LIN {X 0,Y 703.927,Z 1274.734,A -85,B 0,C 180,E1 33383.475,E2 33383.475} C_VEL
LIN {X 0,Y 703.945,Z 1269.075,A -85,B 0,C 180,E1 33381.341,E2 33381.341} C_VEL
LIN {X 0,Y 703.988,Z 1263.047,A -85,B 0,C 180,E1 33379.525,E2 33379.525} C_VEL
LIN {X 0,Y 704.038,Z 1256.148,A -85,B 0,C 180,E1 33377.783,E2 33377.783} C_VEL
LIN {X 0,Y 704.117,Z 1248.477,A -85,B 0,C 180,E1 33376.114,E2 33376.114} C_VEL
LIN {X 0,Y 704.293,Z 1239.669,A -85,B 0,C 180,E1 33374.436,E2 33374.436} C_VEL
LIN {X 0,Y 704.505,Z 1227.564,A -85,B 0,C 180,E1 33372.404,E2 33372.404} C_VEL
LIN {X 0,Y 704.843,Z 1213.387,A -85,B 0,C 180,E1 33370.354,E2 33370.354} C_VEL
LIN {X 0,Y 705.204,Z 1199.968,A -85,B 0,C 180,E1 33368.63,E2 33368.63} C_VEL
LIN {X 0,Y 705.659,Z 1184.756,A -85,B 0,C 180,E1 33366.869,E2 33366.869} C_VEL
LIN {X 0,Y 706.269,Z 1165.244,A -85,B 0,C 180,E1 33364.867,E2 33364.867} C_VEL
LIN {X 0,Y 706.869,Z 1148.784,A -85,B 0,C 180,E1 33363.359,E2 33363.359} C_VEL
LIN {X 0,Y 707.577,Z 1129.955,A -85,B 0,C 180,E1 33361.792,E2 33361.792} C_VEL
LIN {X 0,Y 708.393,Z 1107.88,A -85,B 0,C 180,E1 33360.162,E2 33360.162} C_VEL
LIN {X 0,Y 709.153,Z 1088.525,A -85,B 0,C 180,E1 33358.886,E2 33358.886} C_VEL
LIN {X 0,Y 709.96,Z 1068.119,A -85,B 0,C 180,E1 33357.675,E2 33357.675} C_VEL
LIN {X 0,Y 710.89,Z 1042.665,A -85,B 0,C 180,E1 33356.347,E2 33356.347} C_VEL
LIN {X 0,Y 711.695,Z 1019.844,A -85,B 0,C 180,E1 33355.32,E2 33355.32} C_VEL
LIN {X 0,Y 712.417,Z 998.315,A -85,B 0,C 180,E1 33354.476,E2 33354.476} C_VEL
LIN {X 0,Y 713.159,Z 973.738,A -85,B 0,C 180,E1 33353.65,E2 33353.65} C_VEL
LIN {X 0,Y 713.879,Z 946.765,A -85,B 0,C 180,E1 33352.917,E2 33352.917} C_VEL
LIN {X 0,Y 714.411,Z 921.427,A -85,B 0,C 180,E1 33352.385,E2 33352.385} C_VEL
LIN {X 0,Y 714.824,Z 894.806,A -85,B 0,C 180,E1 33351.976,E2 33351.976} C_VEL
LIN {X 0,Y 716.429,Z 669.278,A -85,B 0,C 180,E1 33349.208,E2 33349.208} C_VEL
LIN {X 0,Y 717.956,Z 467.094,A -85,B 0,C 180,E1 33346.646,E2 33346.646} C_VEL
LIN {X 0,Y 717.985,Z 440.156,A -85,B 0,C 180,E1 33346.285,E2 33346.285} C_VEL
LIN {X 0,Y 714.944,Z 426.613,A -85,B 0,C 180,E1 33345.845,E2 33345.845} C_VEL
LIN {X 0,Y 716.163,Z 384.694,A -85,B 0,C 180,E1 33343.277,E2 33343.277} C_VEL
LIN {X 0,Y 716.843,Z 358.503,A -85,B 0,C 180,E1 33341.602,E2 33341.602} C_VEL
LIN {X 0,Y 710.556,Z 346.163,A -85,B 0,C 180,E1 33340.173,E2 33340.173} C_VEL
LIN {X 0,Y 708.125,Z 341.731,A -85,B 0,C 180,E1 33339.661,E2 33339.661} C_VEL
LIN {X 0,Y 705.926,Z 337.366,A -85,B 0,C 180,E1 33339.178,E2 33339.178} C_VEL
LIN {X 0,Y 704.356,Z 333.75,A -85,B 0,C 180,E1 33338.758,E2 33338.758} C_VEL
LIN {X 0,Y 704.322,Z 333.434,A -85,B 0,C 180,E1 33337.52,E2 33337.52} C_VEL
LIN {X 0,Y 704.318,Z 333.498,A -85,B 0,C 180,E1 33334.574,E2 33334.574} C_VEL
LIN {X 0,Y 704.327,Z 333.497,A -85,B 0,C 180,E1 33331.686,E2 33331.686} C_VEL
LIN {X 0,Y 704.321,Z 333.495,A -85,B 0,C 180,E1 33328.768,E2 33328.768} C_VEL
LIN {X 0,Y 704.338,Z 333.487,A -85,B 0,C 180,E1 33325.838,E2 33325.838} C_VEL
LIN {X 0,Y 704.329,Z 333.5,A -85,B 0,C 180,E1 33322.715,E2 33322.715} C_VEL
LIN {X 0,Y 704.341,Z 333.489,A -85,B 0,C 180,E1 33319.661,E2 33319.661} C_VEL
LIN {X 0,Y 704.329,Z 333.498,A -85,B 0,C 180,E1 33316.58,E2 33316.58} C_VEL
LIN {X 0,Y 704.337,Z 333.489,A -85,B 0,C 180,E1 33313.547,E2 33313.547} C_VEL
LIN {X 0,Y 704.325,Z 333.499,A -85,B 0,C 180,E1 33310.387,E2 33310.387} C_VEL
LIN {X 0,Y 704.326,Z 333.489,A -85,B 0,C 180,E1 33307.423,E2 33307.423} C_VEL
LIN {X 0,Y 704.333,Z 333.498,A -85,B 0,C 180,E1 33304.315,E2 33304.315} C_VEL
LIN {X 0,Y 704.311,Z 333.487,A -85,B 0,C 180,E1 33301.383,E2 33301.383} C_VEL
LIN {X 0,Y 704.339,Z 333.497,A -85,B 0,C 180,E1 33298.373,E2 33298.373} C_VEL
LIN {X 0,Y 704.298,Z 333.494,A -85,B 0,C 180,E1 33295.522,E2 33295.522} C_VEL
LIN {X 0,Y 704.343,Z 333.489,A -85,B 0,C 180,E1 33292.66,E2 33292.66} C_VEL
LIN {X 0,Y 704.306,Z 333.497,A -85,B 0,C 180,E1 33289.613,E2 33289.613} C_VEL
LIN {X 0,Y 704.317,Z 333.49,A -85,B 0,C 180,E1 33286.787,E2 33286.787} C_VEL
LIN {X 0,Y 704.324,Z 333.496,A -85,B 0,C 180,E1 33283.671,E2 33283.671} C_VEL
LIN {X 0,Y 704.296,Z 333.493,A -85,B 0,C 180,E1 33280.855,E2 33280.855} C_VEL
LIN {X 0,Y 704.341,Z 333.492,A -85,B 0,C 180,E1 33278.057,E2 33278.057} C_VEL
LIN {X 0,Y 703.352,Z 333.624,A -85,B 0,C 180,E1 33277.431,E2 33277.431} C_VEL
LIN {X 0,Y 696.918,Z 334.424,A -85,B 0,C 180,E1 33275.675,E2 33275.675} C_VEL
LIN {X 0,Y 696.363,Z 334.487,A -85,B 0,C 180,E1 33275.219,E2 33275.219} C_VEL
LIN {X 0,Y 696.361,Z 334.481,A -85,B 0,C 180,E1 33272.461,E2 33272.461} C_VEL
LIN {X 0,Y 696.403,Z 334.486,A -85,B 0,C 180,E1 33269.451,E2 33269.451} C_VEL
LIN {X 0,Y 696.346,Z 334.484,A -85,B 0,C 180,E1 33266.636,E2 33266.636} C_VEL
LIN {X 0,Y 696.399,Z 334.477,A -85,B 0,C 180,E1 33263.795,E2 33263.795} C_VEL
LIN {X 0,Y 696.358,Z 334.487,A -85,B 0,C 180,E1 33260.817,E2 33260.817} C_VEL
LIN {X 0,Y 696.349,Z 334.481,A -85,B 0,C 180,E1 33258.11,E2 33258.11} C_VEL
LIN {X 0,Y 696.402,Z 334.485,A -85,B 0,C 180,E1 33255.056,E2 33255.056} C_VEL
LIN {X 0,Y 696.338,Z 334.483,A -85,B 0,C 180,E1 33252.222,E2 33252.222} C_VEL
LIN {X 0,Y 696.388,Z 334.481,A -85,B 0,C 180,E1 33249.423,E2 33249.423} C_VEL
LIN {X 0,Y 696.347,Z 334.485,A -85,B 0,C 180,E1 33246.337,E2 33246.337} C_VEL
LIN {X 0,Y 696.336,Z 334.485,A -85,B 0,C 180,E1 33243.756,E2 33243.756} C_VEL
LIN {X 0,Y 696.406,Z 334.484,A -85,B 0,C 180,E1 33240.835,E2 33240.835} C_VEL
LIN {X 0,Y 696.336,Z 334.487,A -85,B 0,C 180,E1 33237.981,E2 33237.981} C_VEL
LIN {X 0,Y 696.336,Z 334.484,A -85,B 0,C 180,E1 33235.417,E2 33235.417} C_VEL
LIN {X 0,Y 696.402,Z 334.485,A -85,B 0,C 180,E1 33232.452,E2 33232.452} C_VEL
LIN {X 0,Y 696.326,Z 334.487,A -85,B 0,C 180,E1 33229.612,E2 33229.612} C_VEL
LIN {X 0,Y 696.34,Z 334.484,A -85,B 0,C 180,E1 33227.033,E2 33227.033} C_VEL
LIN {X 0,Y 696.367,Z 334.489,A -85,B 0,C 180,E1 33223.959,E2 33223.959} C_VEL
LIN {X 0,Y 696.321,Z 334.488,A -85,B 0,C 180,E1 33221.345,E2 33221.345} C_VEL
LIN {X 0,Y 696.33,Z 334.487,A -85,B 0,C 180,E1 33218.838,E2 33218.838} C_VEL
LIN {X 0,Y 696.384,Z 334.487,A -85,B 0,C 180,E1 33215.851,E2 33215.851} C_VEL
LIN {X 0,Y 696.316,Z 334.487,A -85,B 0,C 180,E1 33213.128,E2 33213.128} C_VEL
LIN {X 0,Y 696.32,Z 334.488,A -85,B 0,C 180,E1 33210.658,E2 33210.658} C_VEL
LIN {X 0,Y 696.398,Z 334.477,A -85,B 0,C 180,E1 33207.778,E2 33207.778} C_VEL
LIN {X 0,Y 696.316,Z 334.491,A -85,B 0,C 180,E1 33204.975,E2 33204.975} C_VEL
LIN {X 0,Y 696.307,Z 334.482,A -85,B 0,C 180,E1 33202.575,E2 33202.575} C_VEL
LIN {X 0,Y 696.346,Z 334.488,A -85,B 0,C 180,E1 33199.995,E2 33199.995} C_VEL
LIN {X 0,Y 696.329,Z 334.487,A -85,B 0,C 180,E1 33196.971,E2 33196.971} C_VEL
LIN {X 0,Y 696.297,Z 334.445,A -85,B 0,C 180,E1 33194.487,E2 33194.487} C_VEL
LIN {X 0,Y 696.307,Z 334.497,A -85,B 0,C 180,E1 33192.104,E2 33192.104} C_VEL
LIN {X 0,Y 696.341,Z 334.649,A -85,B 0,C 180,E1 33189.872,E2 33189.872} C_VEL
LIN {X 0,Y 696.737,Z 336.158,A -85,B 0,C 180,E1 33189.711,E2 33189.711} C_VEL
LIN {X 0,Y 698.764,Z 339.241,A -85,B 0,C 180,E1 33189.499,E2 33189.499} C_VEL
LIN {X 0,Y 700.049,Z 340.739,A -85,B 0,C 180,E1 33189.375,E2 33189.375} C_VEL
LIN {X 0,Y 702.798,Z 344.75,A -85,B 0,C 180,E1 33189.1,E2 33189.1} C_VEL
LIN {X 0,Y 711.791,Z 357.759,A -85,B 0,C 180,E1 33188.224,E2 33188.224} C_VEL
LIN {X 0,Y 709.906,Z 574.025,A -85,B 0,C 180,E1 33185.485,E2 33185.485} C_VEL
LIN {X 0,Y 708.338,Z 756.926,A -85,B 0,C 180,E1 33183.213,E2 33183.213} C_VEL
LIN {X 0,Y 707.781,Z 783.361,A -85,B 0,C 180,E1 33182.736,E2 33182.736} C_VEL
LIN {X 0,Y 707.033,Z 810.776,A -85,B 0,C 180,E1 33182.072,E2 33182.072} C_VEL
LIN {X 0,Y 706.205,Z 836.973,A -85,B 0,C 180,E1 33181.27,E2 33181.27} C_VEL
LIN {X 0,Y 705.265,Z 863.108,A -85,B 0,C 180,E1 33180.298,E2 33180.298} C_VEL
LIN {X 0,Y 704.347,Z 885.53,A -85,B 0,C 180,E1 33179.318,E2 33179.318} C_VEL
LIN {X 0,Y 703.388,Z 907.599,A -85,B 0,C 180,E1 33178.221,E2 33178.221} C_VEL
LIN {X 0,Y 702.311,Z 932.34,A -85,B 0,C 180,E1 33176.815,E2 33176.815} C_VEL
LIN {X 0,Y 701.291,Z 954.708,A -85,B 0,C 180,E1 33175.354,E2 33175.354} C_VEL
LIN {X 0,Y 700.372,Z 975.753,A -85,B 0,C 180,E1 33173.82,E2 33173.82} C_VEL
LIN {X 0,Y 699.424,Z 997.558,A -85,B 0,C 180,E1 33172.017,E2 33172.017} C_VEL
LIN {X 0,Y 698.694,Z 1015.217,A -85,B 0,C 180,E1 33170.383,E2 33170.383} C_VEL
LIN {X 0,Y 697.952,Z 1034.923,A -85,B 0,C 180,E1 33168.339,E2 33168.339} C_VEL
LIN {X 0,Y 697.377,Z 1050.921,A -85,B 0,C 180,E1 33166.461,E2 33166.461} C_VEL
LIN {X 0,Y 696.942,Z 1065.694,A -85,B 0,C 180,E1 33164.518,E2 33164.518} C_VEL
LIN {X 0,Y 696.588,Z 1079.58,A -85,B 0,C 180,E1 33162.427,E2 33162.427} C_VEL
LIN {X 0,Y 696.347,Z 1090.39,A -85,B 0,C 180,E1 33160.573,E2 33160.573} C_VEL
LIN {X 0,Y 696.166,Z 1100.117,A -85,B 0,C 180,E1 33158.666,E2 33158.666} C_VEL
LIN {X 0,Y 696.047,Z 1109.981,A -85,B 0,C 180,E1 33156.391,E2 33156.391} C_VEL
LIN {X 0,Y 695.97,Z 1117.369,A -85,B 0,C 180,E1 33154.276,E2 33154.276} C_VEL
LIN {X 0,Y 695.924,Z 1123.234,A -85,B 0,C 180,E1 33152.194,E2 33152.194} C_VEL
LIN {X 0,Y 695.921,Z 1127.907,A -85,B 0,C 180,E1 33149.905,E2 33149.905} C_VEL
LIN {X 0,Y 695.908,Z 1130.641,A -85,B 0,C 180,E1 33147.741,E2 33147.741} C_VEL
LIN {X 0,Y 695.912,Z 1131.788,A -85,B 0,C 180,E1 33145.808,E2 33145.808} C_VEL
LIN {X 0,Y 695.898,Z 1131.751,A -85,B 0,C 180,E1 33143.963,E2 33143.963} C_VEL
LIN {X 0,Y 695.919,Z 1130.287,A -85,B 0,C 180,E1 33141.758,E2 33141.758} C_VEL
LIN {X 0,Y 695.922,Z 1127.061,A -85,B 0,C 180,E1 33139.522,E2 33139.522} C_VEL
LIN {X 0,Y 695.925,Z 1122.434,A -85,B 0,C 180,E1 33137.389,E2 33137.389} C_VEL
LIN {X 0,Y 695.993,Z 1115.61,A -85,B 0,C 180,E1 33135.072,E2 33135.072} C_VEL
LIN {X 0,Y 696.038,Z 1107.302,A -85,B 0,C 180,E1 33132.866,E2 33132.866} C_VEL
LIN {X 0,Y 696.194,Z 1099,A -85,B 0,C 180,E1 33131.012,E2 33131.012} C_VEL
LIN {X 0,Y 696.387,Z 1089.022,A -85,B 0,C 180,E1 33129.087,E2 33129.087} C_VEL
LIN {X 0,Y 696.674,Z 1076.099,A -85,B 0,C 180,E1 33126.924,E2 33126.924} C_VEL
LIN {X 0,Y 697.046,Z 1062.353,A -85,B 0,C 180,E1 33124.937,E2 33124.937} C_VEL
LIN {X 0,Y 697.47,Z 1048.27,A -85,B 0,C 180,E1 33123.123,E2 33123.123} C_VEL
LIN {X 0,Y 698.07,Z 1031.11,A -85,B 0,C 180,E1 33121.149,E2 33121.149} C_VEL
LIN {X 0,Y 698.778,Z 1013.332,A -85,B 0,C 180,E1 33119.344,E2 33119.344} C_VEL
LIN {X 0,Y 699.553,Z 994.517,A -85,B 0,C 180,E1 33117.624,E2 33117.624} C_VEL
LIN {X 0,Y 700.487,Z 972.763,A -85,B 0,C 180,E1 33115.866,E2 33115.866} C_VEL
LIN {X 0,Y 701.376,Z 953.003,A -85,B 0,C 180,E1 33114.437,E2 33114.437} C_VEL
LIN {X 0,Y 702.421,Z 929.574,A -85,B 0,C 180,E1 33112.927,E2 33112.927} C_VEL
LIN {X 0,Y 703.401,Z 907.056,A -85,B 0,C 180,E1 33111.663,E2 33111.663} C_VEL
LIN {X 0,Y 704.332,Z 885.808,A -85,B 0,C 180,E1 33110.604,E2 33110.604} C_VEL
LIN {X 0,Y 705.292,Z 862.464,A -85,B 0,C 180,E1 33109.586,E2 33109.586} C_VEL
LIN {X 0,Y 706.21,Z 835.969,A -85,B 0,C 180,E1 33108.608,E2 33108.608} C_VEL
LIN {X 0,Y 707.023,Z 811.275,A -85,B 0,C 180,E1 33107.851,E2 33107.851} C_VEL
LIN {X 0,Y 707.764,Z 783.948,A -85,B 0,C 180,E1 33107.188,E2 33107.188} C_VEL
LIN {X 0,Y 708.328,Z 757.437,A -85,B 0,C 180,E1 33106.705,E2 33106.705} C_VEL
LIN {X 0,Y 709.316,Z 647.05,A -85,B 0,C 180,E1 33105.331,E2 33105.331} C_VEL
LIN {X 0,Y 711.178,Z 426.373,A -85,B 0,C 180,E1 33102.565,E2 33102.565} C_VEL
LIN {X 0,Y 711.649,Z 357.417,A -85,B 0,C 180,E1 33101.67,E2 33101.67} C_VEL
LIN {X 0,Y 702.078,Z 343.929,A -85,B 0,C 180,E1 33100.742,E2 33100.742} C_VEL
LIN {X 0,Y 699.186,Z 339.581,A -85,B 0,C 180,E1 33100.449,E2 33100.449} C_VEL
LIN {X 0,Y 696.996,Z 336.674,A -85,B 0,C 180,E1 33100.231,E2 33100.231} C_VEL
LIN {X 0,Y 696.462,Z 335.032,A -85,B 0,C 180,E1 33100.108,E2 33100.108} C_VEL
LIN {X 0,Y 696.351,Z 334.473,A -85,B 0,C 180,E1 33099.895,E2 33099.895} C_VEL
LIN {X 0,Y 696.353,Z 334.491,A -85,B 0,C 180,E1 33097.189,E2 33097.189} C_VEL
LIN {X 0,Y 696.4,Z 334.484,A -85,B 0,C 180,E1 33094.188,E2 33094.188} C_VEL
LIN {X 0,Y 696.356,Z 334.488,A -85,B 0,C 180,E1 33091.32,E2 33091.32} C_VEL
LIN {X 0,Y 696.402,Z 334.488,A -85,B 0,C 180,E1 33088.491,E2 33088.491} C_VEL
LIN {X 0,Y 696.375,Z 334.485,A -85,B 0,C 180,E1 33085.504,E2 33085.504} C_VEL
LIN {X 0,Y 696.402,Z 334.487,A -85,B 0,C 180,E1 33082.499,E2 33082.499} C_VEL
LIN {X 0,Y 696.421,Z 334.785,A -85,B 0,C 180,E1 33081.356,E2 33081.356} C_VEL
LIN {X 0,Y 698.749,Z 340.781,A -85,B 0,C 180,E1 33080.872,E2 33080.872} C_VEL
LIN {X 0,Y 701.564,Z 346.305,A -85,B 0,C 180,E1 33080.425,E2 33080.425} C_VEL
LIN {X 0,Y 705.551,Z 352.532,A -85,B 0,C 180,E1 33079.848,E2 33079.848} C_VEL
LIN {X 0,Y 710.85,Z 363.326,A -85,B 0,C 180,E1 33078.615,E2 33078.615} C_VEL
LIN {X 0,Y 709.379,Z 406.198,A -85,B 0,C 180,E1 33075.896,E2 33075.896} C_VEL
LIN {X 0,Y 708.803,Z 427.533,A -85,B 0,C 180,E1 33074.608,E2 33074.608} C_VEL
LIN {X 0,Y 712.341,Z 443.728,A -85,B 0,C 180,E1 33074.102,E2 33074.102} C_VEL
LIN {X 0,Y 710.521,Z 651.598,A -85,B 0,C 180,E1 33071.437,E2 33071.437} C_VEL
LIN {X 0,Y 708.679,Z 876.939,A -85,B 0,C 180,E1 33068.644,E2 33068.644} C_VEL
LIN {X 0,Y 708.246,Z 912.642,A -85,B 0,C 180,E1 33068.168,E2 33068.168} C_VEL
LIN {X 0,Y 707.599,Z 939.832,A -85,B 0,C 180,E1 33067.639,E2 33067.639} C_VEL
LIN {X 0,Y 706.916,Z 964.802,A -85,B 0,C 180,E1 33067.005,E2 33067.005} C_VEL
LIN {X 0,Y 706.06,Z 991.897,A -85,B 0,C 180,E1 33066.144,E2 33066.144} C_VEL
LIN {X 0,Y 705.112,Z 1016.375,A -85,B 0,C 180,E1 33065.205,E2 33065.205} C_VEL
LIN {X 0,Y 704.279,Z 1036.705,A -85,B 0,C 180,E1 33064.307,E2 33064.307} C_VEL
LIN {X 0,Y 703.406,Z 1056.971,A -85,B 0,C 180,E1 33063.296,E2 33063.296} C_VEL
LIN {X 0,Y 702.348,Z 1081.204,A -85,B 0,C 180,E1 33061.929,E2 33061.929} C_VEL
LIN {X 0,Y 701.362,Z 1103.247,A -85,B 0,C 180,E1 33060.499,E2 33060.499} C_VEL
LIN {X 0,Y 700.517,Z 1121.866,A -85,B 0,C 180,E1 33059.156,E2 33059.156} C_VEL
LIN {X 0,Y 699.619,Z 1142.685,A -85,B 0,C 180,E1 33057.492,E2 33057.492} C_VEL
LIN {X 0,Y 698.828,Z 1162.077,A -85,B 0,C 180,E1 33055.728,E2 33055.728} C_VEL
LIN {X 0,Y 698.179,Z 1178.396,A -85,B 0,C 180,E1 33054.089,E2 33054.089} C_VEL
LIN {X 0,Y 697.52,Z 1197.253,A -85,B 0,C 180,E1 33051.955,E2 33051.955} C_VEL
LIN {X 0,Y 697.047,Z 1211.455,A -85,B 0,C 180,E1 33050.137,E2 33050.137} C_VEL
LIN {X 0,Y 696.713,Z 1224.172,A -85,B 0,C 180,E1 33048.318,E2 33048.318} C_VEL
LIN {X 0,Y 696.386,Z 1237.808,A -85,B 0,C 180,E1 33046.088,E2 33046.088} C_VEL
LIN {X 0,Y 696.205,Z 1247.732,A -85,B 0,C 180,E1 33044.201,E2 33044.201} C_VEL
LIN {X 0,Y 696.084,Z 1255.793,A -85,B 0,C 180,E1 33042.443,E2 33042.443} C_VEL
LIN {X 0,Y 695.993,Z 1262.437,A -85,B 0,C 180,E1 33040.764,E2 33040.764} C_VEL
LIN {X 0,Y 695.917,Z 1268.051,A -85,B 0,C 180,E1 33039.093,E2 33039.093} C_VEL
LIN {X 0,Y 695.925,Z 1273.173,A -85,B 0,C 180,E1 33037.264,E2 33037.264} C_VEL
LIN {X 0,Y 695.916,Z 1277.782,A -85,B 0,C 180,E1 33035.028,E2 33035.028} C_VEL
LIN {X 0,Y 695.913,Z 1280.541,A -85,B 0,C 180,E1 33032.882,E2 33032.882} C_VEL
LIN {X 0,Y 695.878,Z 1281.715,A -85,B 0,C 180,E1 33031.07,E2 33031.07} C_VEL
LIN {X 0,Y 695.863,Z 1281.827,A -85,B 0,C 180,E1 33029.341,E2 33029.341} C_VEL
LIN {X 0,Y 695.905,Z 1280.946,A -85,B 0,C 180,E1 33027.612,E2 33027.612} C_VEL
LIN {X 0,Y 695.918,Z 1278.853,A -85,B 0,C 180,E1 33025.666,E2 33025.666} C_VEL
LIN {X 0,Y 695.926,Z 1274.734,A -85,B 0,C 180,E1 33023.4,E2 33023.4} C_VEL
LIN {X 0,Y 695.941,Z 1269.075,A -85,B 0,C 180,E1 33021.24,E2 33021.24} C_VEL
LIN {X 0,Y 695.996,Z 1263.048,A -85,B 0,C 180,E1 33019.404,E2 33019.404} C_VEL
LIN {X 0,Y 696.063,Z 1256.506,A -85,B 0,C 180,E1 33017.725,E2 33017.725} C_VEL
LIN {X 0,Y 696.174,Z 1248.478,A -85,B 0,C 180,E1 33015.953,E2 33015.953} C_VEL
LIN {X 0,Y 696.369,Z 1239.165,A -85,B 0,C 180,E1 33014.161,E2 33014.161} C_VEL
LIN {X 0,Y 696.654,Z 1225.895,A -85,B 0,C 180,E1 33011.94,E2 33011.94} C_VEL
LIN {X 0,Y 697.024,Z 1212.369,A -85,B 0,C 180,E1 33009.986,E2 33009.986} C_VEL
LIN {X 0,Y 697.452,Z 1199.156,A -85,B 0,C 180,E1 33008.279,E2 33008.279} C_VEL
LIN {X 0,Y 698.04,Z 1182.604,A -85,B 0,C 180,E1 33006.355,E2 33006.355} C_VEL
LIN {X 0,Y 698.731,Z 1164.313,A -85,B 0,C 180,E1 33004.486,E2 33004.486} C_VEL
LIN {X 0,Y 699.394,Z 1147.759,A -85,B 0,C 180,E1 33002.959,E2 33002.959} C_VEL
LIN {X 0,Y 700.302,Z 1127.096,A -85,B 0,C 180,E1 33001.239,E2 33001.239} C_VEL
LIN {X 0,Y 701.203,Z 1106.557,A -85,B 0,C 180,E1 32999.73,E2 32999.73} C_VEL
LIN {X 0,Y 702.052,Z 1087.8,A -85,B 0,C 180,E1 32998.487,E2 32998.487} C_VEL
LIN {X 0,Y 702.956,Z 1067.592,A -85,B 0,C 180,E1 32997.282,E2 32997.282} C_VEL
LIN {X 0,Y 704.057,Z 1041.576,A -85,B 0,C 180,E1 32995.922,E2 32995.922} C_VEL
LIN {X 0,Y 704.97,Z 1019.463,A -85,B 0,C 180,E1 32994.924,E2 32994.924} C_VEL
LIN {X 0,Y 705.778,Z 998.318,A -85,B 0,C 180,E1 32994.09,E2 32994.09} C_VEL
LIN {X 0,Y 706.614,Z 973.735,A -85,B 0,C 180,E1 32993.259,E2 32993.259} C_VEL
LIN {X 0,Y 707.452,Z 946.273,A -85,B 0,C 180,E1 32992.51,E2 32992.51} C_VEL
LIN {X 0,Y 708.044,Z 921.116,A -85,B 0,C 180,E1 32991.981,E2 32991.981} C_VEL
LIN {X 0,Y 708.523,Z 894.337,A -85,B 0,C 180,E1 32991.569,E2 32991.569} C_VEL
LIN {X 0,Y 710.368,Z 668.85,A -85,B 0,C 180,E1 32988.779,E2 32988.779} C_VEL
LIN {X 0,Y 712.133,Z 466.713,A -85,B 0,C 180,E1 32986.197,E2 32986.197} C_VEL
LIN {X 0,Y 712.173,Z 442.155,A -85,B 0,C 180,E1 32985.863,E2 32985.863} C_VEL
LIN {X 0,Y 708.699,Z 426.816,A -85,B 0,C 180,E1 32985.363,E2 32985.363} C_VEL
LIN {X 0,Y 710.076,Z 385.529,A -85,B 0,C 180,E1 32982.808,E2 32982.808} C_VEL
LIN {X 0,Y 710.72,Z 362.848,A -85,B 0,C 180,E1 32981.34,E2 32981.34} C_VEL
LIN {X 0,Y 703.259,Z 348.268,A -85,B 0,C 180,E1 32979.672,E2 32979.672} C_VEL
LIN {X 0,Y 700.966,Z 344.115,A -85,B 0,C 180,E1 32979.192,E2 32979.192} C_VEL
LIN {X 0,Y 697.641,Z 337.843,A -85,B 0,C 180,E1 32978.465,E2 32978.465} C_VEL
LIN {X 0,Y 696.424,Z 334.681,A -85,B 0,C 180,E1 32978.075,E2 32978.075} C_VEL
LIN {X 0,Y 696.395,Z 334.468,A -85,B 0,C 180,E1 32975.355,E2 32975.355} C_VEL
LIN {X 0,Y 696.384,Z 334.485,A -85,B 0,C 180,E1 32972.382,E2 32972.382} C_VEL
LIN {X 0,Y 696.391,Z 334.486,A -85,B 0,C 180,E1 32969.363,E2 32969.363} C_VEL
LIN {X 0,Y 696.374,Z 334.481,A -85,B 0,C 180,E1 32966.431,E2 32966.431} C_VEL
LIN {X 0,Y 696.392,Z 334.478,A -85,B 0,C 180,E1 32963.526,E2 32963.526} C_VEL
LIN {X 0,Y 696.384,Z 334.486,A -85,B 0,C 180,E1 32960.586,E2 32960.586} C_VEL
LIN {X 0,Y 696.402,Z 334.474,A -85,B 0,C 180,E1 32957.549,E2 32957.549} C_VEL
LIN {X 0,Y 696.385,Z 334.487,A -85,B 0,C 180,E1 32954.468,E2 32954.468} C_VEL
LIN {X 0,Y 696.396,Z 334.474,A -85,B 0,C 180,E1 32951.428,E2 32951.428} C_VEL
LIN {X 0,Y 696.388,Z 334.485,A -85,B 0,C 180,E1 32948.338,E2 32948.338} C_VEL
LIN {X 0,Y 696.386,Z 334.474,A -85,B 0,C 180,E1 32945.355,E2 32945.355} C_VEL
LIN {X 0,Y 696.391,Z 334.482,A -85,B 0,C 180,E1 32942.222,E2 32942.222} C_VEL
LIN {X 0,Y 696.376,Z 334.48,A -85,B 0,C 180,E1 32939.26,E2 32939.26} C_VEL
LIN {X 0,Y 696.396,Z 334.489,A -85,B 0,C 180,E1 32936.131,E2 32936.131} C_VEL
LIN {X 0,Y 696.363,Z 334.481,A -85,B 0,C 180,E1 32933.238,E2 32933.238} C_VEL
LIN {X 0,Y 696.398,Z 334.483,A -85,B 0,C 180,E1 32930.329,E2 32930.329} C_VEL
LIN {X 0,Y 696.358,Z 334.485,A -85,B 0,C 180,E1 32927.393,E2 32927.393} C_VEL
LIN {X 0,Y 696.4,Z 334.478,A -85,B 0,C 180,E1 32924.511,E2 32924.511} C_VEL
LIN {X 0,Y 696.366,Z 334.487,A -85,B 0,C 180,E1 32921.412,E2 32921.412} C_VEL
LIN {X 0,Y 696.368,Z 334.481,A -85,B 0,C 180,E1 32918.61,E2 32918.61} C_VEL
LIN {X 0,Y 696.389,Z 334.489,A -85,B 0,C 180,E1 32915.484,E2 32915.484} C_VEL
LIN {X 0,Y 696.363,Z 334.487,A -85,B 0,C 180,E1 32915.219,E2 32915.219} C_VEL
LIN {X 0,Y 695.339,Z 334.612,A -85,B 0,C 180,E1 32914.585,E2 32914.585} C_VEL
LIN {X 0,Y 688.926,Z 335.409,A -85,B 0,C 180,E1 32912.809,E2 32912.809} C_VEL
LIN {X 0,Y 688.432,Z 335.47,A -85,B 0,C 180,E1 32912.347,E2 32912.347} C_VEL
LIN {X 0,Y 688.432,Z 335.477,A -85,B 0,C 180,E1 32909.156,E2 32909.156} C_VEL
LIN {X 0,Y 688.412,Z 335.472,A -85,B 0,C 180,E1 32906.4,E2 32906.4} C_VEL
LIN {X 0,Y 688.465,Z 335.471,A -85,B 0,C 180,E1 32903.431,E2 32903.431} C_VEL
LIN {X 0,Y 688.407,Z 335.474,A -85,B 0,C 180,E1 32900.597,E2 32900.597} C_VEL
LIN {X 0,Y 688.43,Z 335.468,A -85,B 0,C 180,E1 32897.854,E2 32897.854} C_VEL
LIN {X 0,Y 688.428,Z 335.476,A -85,B 0,C 180,E1 32894.746,E2 32894.746} C_VEL
LIN {X 0,Y 688.401,Z 335.471,A -85,B 0,C 180,E1 32892.035,E2 32892.035} C_VEL
LIN {X 0,Y 688.466,Z 335.474,A -85,B 0,C 180,E1 32889.073,E2 32889.073} C_VEL
LIN {X 0,Y 688.398,Z 335.473,A -85,B 0,C 180,E1 32886.136,E2 32886.136} C_VEL
LIN {X 0,Y 688.414,Z 335.473,A -85,B 0,C 180,E1 32883.499,E2 32883.499} C_VEL
LIN {X 0,Y 688.425,Z 335.475,A -85,B 0,C 180,E1 32880.36,E2 32880.36} C_VEL
LIN {X 0,Y 688.391,Z 335.474,A -85,B 0,C 180,E1 32877.697,E2 32877.697} C_VEL
LIN {X 0,Y 688.45,Z 335.47,A -85,B 0,C 180,E1 32874.909,E2 32874.909} C_VEL
LIN {X 0,Y 688.401,Z 335.476,A -85,B 0,C 180,E1 32871.918,E2 32871.918} C_VEL
LIN {X 0,Y 688.389,Z 335.475,A -85,B 0,C 180,E1 32869.34,E2 32869.34} C_VEL
LIN {X 0,Y 688.468,Z 335.473,A -85,B 0,C 180,E1 32866.451,E2 32866.451} C_VEL
LIN {X 0,Y 688.388,Z 335.477,A -85,B 0,C 180,E1 32863.524,E2 32863.524} C_VEL
LIN {X 0,Y 688.389,Z 335.476,A -85,B 0,C 180,E1 32860.969,E2 32860.969} C_VEL
LIN {X 0,Y 688.461,Z 335.475,A -85,B 0,C 180,E1 32858.015,E2 32858.015} C_VEL
LIN {X 0,Y 688.381,Z 335.474,A -85,B 0,C 180,E1 32855.25,E2 32855.25} C_VEL
LIN {X 0,Y 688.381,Z 335.475,A -85,B 0,C 180,E1 32852.747,E2 32852.747} C_VEL
LIN {X 0,Y 688.465,Z 335.474,A -85,B 0,C 180,E1 32849.834,E2 32849.834} C_VEL
LIN {X 0,Y 688.375,Z 335.467,A -85,B 0,C 180,E1 32847.003,E2 32847.003} C_VEL
LIN {X 0,Y 688.372,Z 335.479,A -85,B 0,C 180,E1 32844.582,E2 32844.582} C_VEL
LIN {X 0,Y 688.46,Z 335.468,A -85,B 0,C 180,E1 32841.733,E2 32841.733} C_VEL
LIN {X 0,Y 688.372,Z 335.473,A -85,B 0,C 180,E1 32838.776,E2 32838.776} C_VEL
LIN {X 0,Y 688.367,Z 335.474,A -85,B 0,C 180,E1 32836.352,E2 32836.352} C_VEL
LIN {X 0,Y 688.423,Z 335.43,A -85,B 0,C 180,E1 32833.634,E2 32833.634} C_VEL
LIN {X 0,Y 688.375,Z 335.47,A -85,B 0,C 180,E1 32830.66,E2 32830.66} C_VEL
LIN {X 0,Y 688.46,Z 336.065,A -85,B 0,C 180,E1 32830.442,E2 32830.442} C_VEL
LIN {X 0,Y 690.047,Z 339.453,A -85,B 0,C 180,E1 32830.213,E2 32830.213} C_VEL
LIN {X 0,Y 692.175,Z 341.822,A -85,B 0,C 180,E1 32830.002,E2 32830.002} C_VEL
LIN {X 0,Y 694.989,Z 345.803,A -85,B 0,C 180,E1 32829.713,E2 32829.713} C_VEL
LIN {X 0,Y 705.919,Z 361.525,A -85,B 0,C 180,E1 32828.623,E2 32828.623} C_VEL
LIN {X 0,Y 703.786,Z 577.533,A -85,B 0,C 180,E1 32825.866,E2 32825.866} C_VEL
LIN {X 0,Y 702.045,Z 757.004,A -85,B 0,C 180,E1 32823.618,E2 32823.618} C_VEL
LIN {X 0,Y 701.409,Z 783.465,A -85,B 0,C 180,E1 32823.138,E2 32823.138} C_VEL
LIN {X 0,Y 700.578,Z 810.816,A -85,B 0,C 180,E1 32822.471,E2 32822.471} C_VEL
LIN {X 0,Y 699.62,Z 837.456,A -85,B 0,C 180,E1 32821.651,E2 32821.651} C_VEL
LIN {X 0,Y 698.543,Z 863.777,A -85,B 0,C 180,E1 32820.66,E2 32820.66} C_VEL
LIN {X 0,Y 697.495,Z 886.516,A -85,B 0,C 180,E1 32819.655,E2 32819.655} C_VEL
LIN {X 0,Y 696.373,Z 909.586,A -85,B 0,C 180,E1 32818.49,E2 32818.49} C_VEL
LIN {X 0,Y 695.078,Z 935.142,A -85,B 0,C 180,E1 32817,E2 32817} C_VEL
LIN {X 0,Y 694.035,Z 955.608,A -85,B 0,C 180,E1 32815.641,E2 32815.641} C_VEL
LIN {X 0,Y 692.959,Z 977.255,A -85,B 0,C 180,E1 32814.037,E2 32814.037} C_VEL
LIN {X 0,Y 691.905,Z 998.322,A -85,B 0,C 180,E1 32812.266,E2 32812.266} C_VEL
LIN {X 0,Y 691.069,Z 1016.394,A -85,B 0,C 180,E1 32810.568,E2 32810.568} C_VEL
LIN {X 0,Y 690.229,Z 1035.535,A -85,B 0,C 180,E1 32808.546,E2 32808.546} C_VEL
LIN {X 0,Y 689.593,Z 1051.374,A -85,B 0,C 180,E1 32806.659,E2 32806.659} C_VEL
LIN {X 0,Y 689.064,Z 1067.018,A -85,B 0,C 180,E1 32804.564,E2 32804.564} C_VEL
LIN {X 0,Y 688.665,Z 1080.593,A -85,B 0,C 180,E1 32802.466,E2 32802.466} C_VEL
LIN {X 0,Y 688.359,Z 1092.132,A -85,B 0,C 180,E1 32800.436,E2 32800.436} C_VEL
LIN {X 0,Y 688.169,Z 1103.315,A -85,B 0,C 180,E1 32798.135,E2 32798.135} C_VEL
LIN {X 0,Y 688.018,Z 1111.693,A -85,B 0,C 180,E1 32796.057,E2 32796.057} C_VEL
LIN {X 0,Y 687.972,Z 1118.161,A -85,B 0,C 180,E1 32794.126,E2 32794.126} C_VEL
LIN {X 0,Y 687.931,Z 1123.788,A -85,B 0,C 180,E1 32792.041,E2 32792.041} C_VEL
LIN {X 0,Y 687.916,Z 1128.149,A -85,B 0,C 180,E1 32789.804,E2 32789.804} C_VEL
LIN {X 0,Y 687.905,Z 1130.688,A -85,B 0,C 180,E1 32787.719,E2 32787.719} C_VEL
LIN {X 0,Y 687.909,Z 1131.805,A -85,B 0,C 180,E1 32785.76,E2 32785.76} C_VEL
LIN {X 0,Y 687.909,Z 1131.721,A -85,B 0,C 180,E1 32783.834,E2 32783.834} C_VEL
LIN {X 0,Y 687.918,Z 1130.033,A -85,B 0,C 180,E1 32781.487,E2 32781.487} C_VEL
LIN {X 0,Y 687.922,Z 1126.468,A -85,B 0,C 180,E1 32779.134,E2 32779.134} C_VEL
LIN {X 0,Y 687.92,Z 1121.39,A -85,B 0,C 180,E1 32776.9,E2 32776.9} C_VEL
LIN {X 0,Y 687.978,Z 1114.207,A -85,B 0,C 180,E1 32774.549,E2 32774.549} C_VEL
LIN {X 0,Y 688.069,Z 1106.745,A -85,B 0,C 180,E1 32772.59,E2 32772.59} C_VEL
LIN {X 0,Y 688.247,Z 1098.782,A -85,B 0,C 180,E1 32770.802,E2 32770.802} C_VEL
LIN {X 0,Y 688.464,Z 1088.336,A -85,B 0,C 180,E1 32768.772,E2 32768.772} C_VEL
LIN {X 0,Y 688.845,Z 1074.167,A -85,B 0,C 180,E1 32766.417,E2 32766.417} C_VEL
LIN {X 0,Y 689.284,Z 1060.833,A -85,B 0,C 180,E1 32764.493,E2 32764.493} C_VEL
LIN {X 0,Y 689.823,Z 1045.94,A -85,B 0,C 180,E1 32762.575,E2 32762.575} C_VEL
LIN {X 0,Y 690.569,Z 1027.612,A -85,B 0,C 180,E1 32760.498,E2 32760.498} C_VEL
LIN {X 0,Y 691.358,Z 1009.55,A -85,B 0,C 180,E1 32758.674,E2 32758.674} C_VEL
LIN {X 0,Y 692.402,Z 988.237,A -85,B 0,C 180,E1 32756.771,E2 32756.771} C_VEL
LIN {X 0,Y 693.353,Z 969.018,A -85,B 0,C 180,E1 32755.243,E2 32755.243} C_VEL
LIN {X 0,Y 694.534,Z 945.798,A -85,B 0,C 180,E1 32753.594,E2 32753.594} C_VEL
LIN {X 0,Y 695.725,Z 922.558,A -85,B 0,C 180,E1 32752.153,E2 32752.153} C_VEL
LIN {X 0,Y 696.763,Z 901.606,A -85,B 0,C 180,E1 32751.001,E2 32751.001} C_VEL
LIN {X 0,Y 697.961,Z 876.001,A -85,B 0,C 180,E1 32749.768,E2 32749.768} C_VEL
LIN {X 0,Y 699.066,Z 850.784,A -85,B 0,C 180,E1 32748.741,E2 32748.741} C_VEL
LIN {X 0,Y 699.928,Z 828.298,A -85,B 0,C 180,E1 32747.961,E2 32747.961} C_VEL
LIN {X 0,Y 700.848,Z 802.267,A -85,B 0,C 180,E1 32747.211,E2 32747.211} C_VEL
LIN {X 0,Y 701.619,Z 775.964,A -85,B 0,C 180,E1 32746.62,E2 32746.62} C_VEL
LIN {X 0,Y 702.164,Z 749.874,A -85,B 0,C 180,E1 32746.192,E2 32746.192} C_VEL
LIN {X 0,Y 704.324,Z 522.018,A -85,B 0,C 180,E1 32743.345,E2 32743.345} C_VEL
LIN {X 0,Y 705.79,Z 361.065,A -85,B 0,C 180,E1 32741.271,E2 32741.271} C_VEL
LIN {X 0,Y 694.535,Z 345.283,A -85,B 0,C 180,E1 32740.153,E2 32740.153} C_VEL
LIN {X 0,Y 691.344,Z 340.698,A -85,B 0,C 180,E1 32739.823,E2 32739.823} C_VEL
LIN {X 0,Y 689.055,Z 337.772,A -85,B 0,C 180,E1 32739.589,E2 32739.589} C_VEL
LIN {X 0,Y 688.504,Z 336.091,A -85,B 0,C 180,E1 32739.468,E2 32739.468} C_VEL
LIN {X 0,Y 688.407,Z 335.463,A -85,B 0,C 180,E1 32739.243,E2 32739.243} C_VEL
LIN {X 0,Y 688.465,Z 335.475,A -85,B 0,C 180,E1 32736.278,E2 32736.278} C_VEL
LIN {X 0,Y 688.413,Z 335.477,A -85,B 0,C 180,E1 32733.426,E2 32733.426} C_VEL
LIN {X 0,Y 688.465,Z 335.477,A -85,B 0,C 180,E1 32730.601,E2 32730.601} C_VEL
LIN {X 0,Y 688.433,Z 335.474,A -85,B 0,C 180,E1 32727.548,E2 32727.548} C_VEL
LIN {X 0,Y 688.463,Z 335.478,A -85,B 0,C 180,E1 32724.563,E2 32724.563} C_VEL
LIN {X 0,Y 688.502,Z 335.746,A -85,B 0,C 180,E1 32721.771,E2 32721.771} C_VEL
LIN {X 0,Y 690.256,Z 340.511,A -85,B 0,C 180,E1 32721.366,E2 32721.366} C_VEL
LIN {X 0,Y 695.175,Z 350.997,A -85,B 0,C 180,E1 32720.525,E2 32720.525} C_VEL
LIN {X 0,Y 701.268,Z 360.848,A -85,B 0,C 180,E1 32719.659,E2 32719.659} C_VEL
LIN {X 0,Y 704.774,Z 367.637,A -85,B 0,C 180,E1 32718.88,E2 32718.88} C_VEL
LIN {X 0,Y 703.126,Z 410.083,A -85,B 0,C 180,E1 32716.168,E2 32716.168} C_VEL
LIN {X 0,Y 702.61,Z 427.569,A -85,B 0,C 180,E1 32715.108,E2 32715.108} C_VEL
LIN {X 0,Y 706.566,Z 445.689,A -85,B 0,C 180,E1 32714.53,E2 32714.53} C_VEL
LIN {X 0,Y 704.503,Z 652.87,A -85,B 0,C 180,E1 32711.854,E2 32711.854} C_VEL
LIN {X 0,Y 702.415,Z 877.957,A -85,B 0,C 180,E1 32709.04,E2 32709.04} C_VEL
LIN {X 0,Y 701.921,Z 913.198,A -85,B 0,C 180,E1 32708.565,E2 32708.565} C_VEL
LIN {X 0,Y 701.211,Z 939.991,A -85,B 0,C 180,E1 32708.038,E2 32708.038} C_VEL
LIN {X 0,Y 700.439,Z 964.677,A -85,B 0,C 180,E1 32707.408,E2 32707.408} C_VEL
LIN {X 0,Y 699.445,Z 992.432,A -85,B 0,C 180,E1 32706.52,E2 32706.52} C_VEL
LIN {X 0,Y 698.458,Z 1015.354,A -85,B 0,C 180,E1 32705.636,E2 32705.636} C_VEL
LIN {X 0,Y 697.528,Z 1035.615,A -85,B 0,C 180,E1 32704.741,E2 32704.741} C_VEL
LIN {X 0,Y 696.562,Z 1055.54,A -85,B 0,C 180,E1 32703.746,E2 32703.746} C_VEL
LIN {X 0,Y 695.55,Z 1075.916,A -85,B 0,C 180,E1 32702.604,E2 32702.604} C_VEL
LIN {X 0,Y 694.272,Z 1100.707,A -85,B 0,C 180,E1 32701.027,E2 32701.027} C_VEL
LIN {X 0,Y 693.299,Z 1119.84,A -85,B 0,C 180,E1 32699.648,E2 32699.648} C_VEL
LIN {X 0,Y 692.448,Z 1137.319,A -85,B 0,C 180,E1 32698.256,E2 32698.256} C_VEL
LIN {X 0,Y 691.466,Z 1157.483,A -85,B 0,C 180,E1 32696.478,E2 32696.478} C_VEL
LIN {X 0,Y 690.678,Z 1174.983,A -85,B 0,C 180,E1 32694.732,E2 32694.732} C_VEL
LIN {X 0,Y 690.021,Z 1190.407,A -85,B 0,C 180,E1 32693.032,E2 32693.032} C_VEL
LIN {X 0,Y 689.384,Z 1207.589,A -85,B 0,C 180,E1 32690.903,E2 32690.903} C_VEL
LIN {X 0,Y 688.937,Z 1221.262,A -85,B 0,C 180,E1 32688.971,E2 32688.971} C_VEL
LIN {X 0,Y 688.605,Z 1232.792,A -85,B 0,C 180,E1 32687.143,E2 32687.143} C_VEL
LIN {X 0,Y 688.322,Z 1244.786,A -85,B 0,C 180,E1 32684.98,E2 32684.98} C_VEL
LIN {X 0,Y 688.139,Z 1255.079,A -85,B 0,C 180,E1 32682.759,E2 32682.759} C_VEL
LIN {X 0,Y 688.013,Z 1262.132,A -85,B 0,C 180,E1 32680.975,E2 32680.975} C_VEL
LIN {X 0,Y 687.924,Z 1267.822,A -85,B 0,C 180,E1 32679.276,E2 32679.276} C_VEL
LIN {X 0,Y 687.92,Z 1272.964,A -85,B 0,C 180,E1 32677.433,E2 32677.433} C_VEL
LIN {X 0,Y 687.914,Z 1277.486,A -85,B 0,C 180,E1 32675.254,E2 32675.254} C_VEL
LIN {X 0,Y 687.909,Z 1280.423,A -85,B 0,C 180,E1 32673.061,E2 32673.061} C_VEL
LIN {X 0,Y 687.88,Z 1281.715,A -85,B 0,C 180,E1 32671.083,E2 32671.083} C_VEL
LIN {X 0,Y 687.863,Z 1281.827,A -85,B 0,C 180,E1 32669.334,E2 32669.334} C_VEL
LIN {X 0,Y 687.904,Z 1280.946,A -85,B 0,C 180,E1 32667.584,E2 32667.584} C_VEL
LIN {X 0,Y 687.916,Z 1278.892,A -85,B 0,C 180,E1 32665.643,E2 32665.643} C_VEL
LIN {X 0,Y 687.927,Z 1274.734,A -85,B 0,C 180,E1 32663.323,E2 32663.323} C_VEL
LIN {X 0,Y 687.939,Z 1269.076,A -85,B 0,C 180,E1 32661.137,E2 32661.137} C_VEL
LIN {X 0,Y 688.005,Z 1263.049,A -85,B 0,C 180,E1 32659.279,E2 32659.279} C_VEL
LIN {X 0,Y 688.111,Z 1256.15,A -85,B 0,C 180,E1 32657.496,E2 32657.496} C_VEL
LIN {X 0,Y 688.255,Z 1248.062,A -85,B 0,C 180,E1 32655.7,E2 32655.7} C_VEL
LIN {X 0,Y 688.461,Z 1237.811,A -85,B 0,C 180,E1 32653.722,E2 32653.722} C_VEL
LIN {X 0,Y 688.859,Z 1223.831,A -85,B 0,C 180,E1 32651.414,E2 32651.414} C_VEL
LIN {X 0,Y 689.237,Z 1211.144,A -85,B 0,C 180,E1 32649.582,E2 32649.582} C_VEL
LIN {X 0,Y 689.773,Z 1197.13,A -85,B 0,C 180,E1 32647.769,E2 32647.769} C_VEL
LIN {X 0,Y 690.542,Z 1178.267,A -85,B 0,C 180,E1 32645.614,E2 32645.614} C_VEL
LIN {X 0,Y 691.248,Z 1162.451,A -85,B 0,C 180,E1 32644.006,E2 32644.006} C_VEL
LIN {X 0,Y 692.121,Z 1143.705,A -85,B 0,C 180,E1 32642.278,E2 32642.278} C_VEL
LIN {X 0,Y 693.134,Z 1123.247,A -85,B 0,C 180,E1 32640.612,E2 32640.612} C_VEL
LIN {X 0,Y 694.089,Z 1104.571,A -85,B 0,C 180,E1 32639.243,E2 32639.243} C_VEL
LIN {X 0,Y 695.097,Z 1084.503,A -85,B 0,C 180,E1 32637.917,E2 32637.917} C_VEL
LIN {X 0,Y 696.384,Z 1059.099,A -85,B 0,C 180,E1 32636.442,E2 32636.442} C_VEL
LIN {X 0,Y 697.398,Z 1038.245,A -85,B 0,C 180,E1 32635.384,E2 32635.384} C_VEL
LIN {X 0,Y 698.296,Z 1018.733,A -85,B 0,C 180,E1 32634.505,E2 32634.505} C_VEL
LIN {X 0,Y 699.168,Z 998.316,A -85,B 0,C 180,E1 32633.697,E2 32633.697} C_VEL
LIN {X 0,Y 700.073,Z 974.472,A -85,B 0,C 180,E1 32632.884,E2 32632.884} C_VEL
LIN {X 0,Y 701.017,Z 947.261,A -85,B 0,C 180,E1 32632.131,E2 32632.131} C_VEL
LIN {X 0,Y 701.692,Z 921.903,A -85,B 0,C 180,E1 32631.59,E2 32631.59} C_VEL
LIN {X 0,Y 702.223,Z 896.049,A -85,B 0,C 180,E1 32631.185,E2 32631.185} C_VEL
LIN {X 0,Y 704.325,Z 670.677,A -85,B 0,C 180,E1 32628.372,E2 32628.372} C_VEL
LIN {X 0,Y 706.329,Z 468.645,A -85,B 0,C 180,E1 32625.771,E2 32625.771} C_VEL
LIN {X 0,Y 706.419,Z 444.29,A -85,B 0,C 180,E1 32625.439,E2 32625.439} C_VEL
LIN {X 0,Y 702.502,Z 426.825,A -85,B 0,C 180,E1 32624.862,E2 32624.862} C_VEL
LIN {X 0,Y 704.045,Z 386.084,A -85,B 0,C 180,E1 32622.313,E2 32622.313} C_VEL
LIN {X 0,Y 704.626,Z 367.159,A -85,B 0,C 180,E1 32621.073,E2 32621.073} C_VEL
LIN {X 0,Y 697.529,Z 353.637,A -85,B 0,C 180,E1 32619.529,E2 32619.529} C_VEL
LIN {X 0,Y 689.845,Z 339.035,A -85,B 0,C 180,E1 32617.821,E2 32617.821} C_VEL
LIN {X 0,Y 688.489,Z 335.679,A -85,B 0,C 180,E1 32617.402,E2 32617.402} C_VEL
LIN {X 0,Y 688.443,Z 335.432,A -85,B 0,C 180,E1 32615.825,E2 32615.825} C_VEL
LIN {X 0,Y 688.445,Z 335.474,A -85,B 0,C 180,E1 32612.901,E2 32612.901} C_VEL
LIN {X 0,Y 688.462,Z 335.471,A -85,B 0,C 180,E1 32609.878,E2 32609.878} C_VEL
LIN {X 0,Y 688.452,Z 335.471,A -85,B 0,C 180,E1 32606.852,E2 32606.852} C_VEL
LIN {X 0,Y 688.462,Z 335.464,A -85,B 0,C 180,E1 32603.799,E2 32603.799} C_VEL
LIN {X 0,Y 688.45,Z 335.473,A -85,B 0,C 180,E1 32600.667,E2 32600.667} C_VEL
LIN {X 0,Y 688.463,Z 335.463,A -85,B 0,C 180,E1 32597.583,E2 32597.583} C_VEL
LIN {X 0,Y 688.446,Z 335.475,A -85,B 0,C 180,E1 32594.466,E2 32594.466} C_VEL
LIN {X 0,Y 688.454,Z 335.463,A -85,B 0,C 180,E1 32591.477,E2 32591.477} C_VEL
LIN {X 0,Y 688.45,Z 335.472,A -85,B 0,C 180,E1 32588.351,E2 32588.351} C_VEL
LIN {X 0,Y 688.448,Z 335.463,A -85,B 0,C 180,E1 32585.333,E2 32585.333} C_VEL
LIN {X 0,Y 688.447,Z 335.47,A -85,B 0,C 180,E1 32582.164,E2 32582.164} C_VEL
LIN {X 0,Y 688.445,Z 335.468,A -85,B 0,C 180,E1 32579.168,E2 32579.168} C_VEL
LIN {X 0,Y 688.446,Z 335.476,A -85,B 0,C 180,E1 32576.002,E2 32576.002} C_VEL
LIN {X 0,Y 688.434,Z 335.468,A -85,B 0,C 180,E1 32573.076,E2 32573.076} C_VEL
LIN {X 0,Y 688.458,Z 335.477,A -85,B 0,C 180,E1 32569.96,E2 32569.96} C_VEL
LIN {X 0,Y 688.423,Z 335.471,A -85,B 0,C 180,E1 32567.051,E2 32567.051} C_VEL
LIN {X 0,Y 688.461,Z 335.472,A -85,B 0,C 180,E1 32564.154,E2 32564.154} C_VEL
LIN {X 0,Y 688.42,Z 335.474,A -85,B 0,C 180,E1 32561.259,E2 32561.259} C_VEL
LIN {X 0,Y 688.455,Z 335.468,A -85,B 0,C 180,E1 32558.352,E2 32558.352} C_VEL
LIN {X 0,Y 688.428,Z 335.476,A -85,B 0,C 180,E1 32555.273,E2 32555.273} C_VEL
LIN {X 0,Y 688.42,Z 335.471,A -85,B 0,C 180,E1 32552.492,E2 32552.492} C_VEL
LIN {X 0,Y 688.432,Z 335.47,A -85,B 0,C 180,E1 32552.347,E2 32552.347} C_VEL
LIN {X 0,Y 687.496,Z 335.596,A -85,B 0,C 180,E1 32551.706,E2 32551.706} C_VEL
LIN {X 0,Y 680.988,Z 336.398,A -85,B 0,C 180,E1 32549.864,E2 32549.864} C_VEL
LIN {X 0,Y 680.524,Z 336.463,A -85,B 0,C 180,E1 32549.443,E2 32549.443} C_VEL
LIN {X 0,Y 680.469,Z 336.462,A -85,B 0,C 180,E1 32546.562,E2 32546.562} C_VEL
LIN {X 0,Y 680.526,Z 336.456,A -85,B 0,C 180,E1 32543.626,E2 32543.626} C_VEL
LIN {X 0,Y 680.469,Z 336.463,A -85,B 0,C 180,E1 32540.615,E2 32540.615} C_VEL
LIN {X 0,Y 680.495,Z 336.457,A -85,B 0,C 180,E1 32537.817,E2 32537.817} C_VEL
LIN {X 0,Y 680.481,Z 336.465,A -85,B 0,C 180,E1 32534.668,E2 32534.668} C_VEL
LIN {X 0,Y 680.465,Z 336.459,A -85,B 0,C 180,E1 32531.957,E2 32531.957} C_VEL
LIN {X 0,Y 680.528,Z 336.462,A -85,B 0,C 180,E1 32528.965,E2 32528.965} C_VEL
LIN {X 0,Y 680.458,Z 336.462,A -85,B 0,C 180,E1 32526.08,E2 32526.08} C_VEL
LIN {X 0,Y 680.493,Z 336.461,A -85,B 0,C 180,E1 32523.335,E2 32523.335} C_VEL
LIN {X 0,Y 680.473,Z 336.463,A -85,B 0,C 180,E1 32520.23,E2 32520.23} C_VEL
LIN {X 0,Y 680.456,Z 336.463,A -85,B 0,C 180,E1 32517.572,E2 32517.572} C_VEL
LIN {X 0,Y 680.529,Z 336.462,A -85,B 0,C 180,E1 32514.662,E2 32514.662} C_VEL
LIN {X 0,Y 680.453,Z 336.464,A -85,B 0,C 180,E1 32511.734,E2 32511.734} C_VEL
LIN {X 0,Y 680.463,Z 336.463,A -85,B 0,C 180,E1 32509.118,E2 32509.118} C_VEL
LIN {X 0,Y 680.491,Z 336.465,A -85,B 0,C 180,E1 32506.036,E2 32506.036} C_VEL
LIN {X 0,Y 680.444,Z 336.465,A -85,B 0,C 180,E1 32503.338,E2 32503.338} C_VEL
LIN {X 0,Y 680.477,Z 336.464,A -85,B 0,C 180,E1 32500.669,E2 32500.669} C_VEL
LIN {X 0,Y 680.457,Z 336.466,A -85,B 0,C 180,E1 32497.515,E2 32497.515} C_VEL
LIN {X 0,Y 680.439,Z 336.462,A -85,B 0,C 180,E1 32494.974,E2 32494.974} C_VEL
LIN {X 0,Y 680.502,Z 336.462,A -85,B 0,C 180,E1 32492.189,E2 32492.189} C_VEL
LIN {X 0,Y 680.45,Z 336.468,A -85,B 0,C 180,E1 32489.242,E2 32489.242} C_VEL
LIN {X 0,Y 680.433,Z 336.456,A -85,B 0,C 180,E1 32486.715,E2 32486.715} C_VEL
LIN {X 0,Y 680.499,Z 336.46,A -85,B 0,C 180,E1 32483.927,E2 32483.927} C_VEL
LIN {X 0,Y 680.44,Z 336.469,A -85,B 0,C 180,E1 32480.929,E2 32480.929} C_VEL
LIN {X 0,Y 680.431,Z 336.465,A -85,B 0,C 180,E1 32478.386,E2 32478.386} C_VEL
LIN {X 0,Y 680.511,Z 336.416,A -85,B 0,C 180,E1 32475.532,E2 32475.532} C_VEL
LIN {X 0,Y 680.431,Z 336.454,A -85,B 0,C 180,E1 32472.644,E2 32472.644} C_VEL
LIN {X 0,Y 680.536,Z 336.719,A -85,B 0,C 180,E1 32471.16,E2 32471.16} C_VEL
LIN {X 0,Y 680.85,Z 338.061,A -85,B 0,C 180,E1 32471.025,E2 32471.025} C_VEL
LIN {X 0,Y 682.816,Z 341.192,A -85,B 0,C 180,E1 32470.803,E2 32470.803} C_VEL
LIN {X 0,Y 684.213,Z 342.753,A -85,B 0,C 180,E1 32470.66,E2 32470.66} C_VEL
LIN {X 0,Y 686.88,Z 346.657,A -85,B 0,C 180,E1 32470.375,E2 32470.375} C_VEL
LIN {X 0,Y 695.17,Z 358.277,A -85,B 0,C 180,E1 32469.521,E2 32469.521} C_VEL
LIN {X 0,Y 700.077,Z 365.583,A -85,B 0,C 180,E1 32469.024,E2 32469.024} C_VEL
LIN {X 0,Y 697.694,Z 581.434,A -85,B 0,C 180,E1 32466.248,E2 32466.248} C_VEL
LIN {X 0,Y 695.789,Z 757.072,A -85,B 0,C 180,E1 32464.03,E2 32464.03} C_VEL
LIN {X 0,Y 695.077,Z 783.365,A -85,B 0,C 180,E1 32463.551,E2 32463.551} C_VEL
LIN {X 0,Y 694.157,Z 810.855,A -85,B 0,C 180,E1 32462.878,E2 32462.878} C_VEL
LIN {X 0,Y 693.094,Z 837.202,A -85,B 0,C 180,E1 32462.064,E2 32462.064} C_VEL
LIN {X 0,Y 691.867,Z 864.085,A -85,B 0,C 180,E1 32461.044,E2 32461.044} C_VEL
LIN {X 0,Y 690.713,Z 886.663,A -85,B 0,C 180,E1 32460.038,E2 32460.038} C_VEL
LIN {X 0,Y 689.422,Z 910.581,A -85,B 0,C 180,E1 32458.818,E2 32458.818} C_VEL
LIN {X 0,Y 688.005,Z 935.092,A -85,B 0,C 180,E1 32457.373,E2 32457.373} C_VEL
LIN {X 0,Y 686.86,Z 955.387,A -85,B 0,C 180,E1 32456.014,E2 32456.014} C_VEL
LIN {X 0,Y 685.632,Z 977.393,A -85,B 0,C 180,E1 32454.366,E2 32454.366} C_VEL
LIN {X 0,Y 684.426,Z 998.488,A -85,B 0,C 180,E1 32452.574,E2 32452.574} C_VEL
LIN {X 0,Y 683.491,Z 1016.75,A -85,B 0,C 180,E1 32450.837,E2 32450.837} C_VEL
LIN {X 0,Y 682.543,Z 1035.355,A -85,B 0,C 180,E1 32448.85,E2 32448.85} C_VEL
LIN {X 0,Y 681.829,Z 1051.588,A -85,B 0,C 180,E1 32446.893,E2 32446.893} C_VEL
LIN {X 0,Y 681.217,Z 1067.455,A -85,B 0,C 180,E1 32444.732,E2 32444.732} C_VEL
LIN {X 0,Y 680.774,Z 1080.635,A -85,B 0,C 180,E1 32442.669,E2 32442.669} C_VEL
LIN {X 0,Y 680.445,Z 1092.162,A -85,B 0,C 180,E1 32440.615,E2 32440.615} C_VEL
LIN {X 0,Y 680.201,Z 1103.559,A -85,B 0,C 180,E1 32438.234,E2 32438.234} C_VEL
LIN {X 0,Y 680.04,Z 1111.908,A -85,B 0,C 180,E1 32436.129,E2 32436.129} C_VEL
LIN {X 0,Y 679.978,Z 1118.507,A -85,B 0,C 180,E1 32434.12,E2 32434.12} C_VEL
LIN {X 0,Y 679.932,Z 1124.189,A -85,B 0,C 180,E1 32431.95,E2 32431.95} C_VEL
LIN {X 0,Y 679.917,Z 1128.231,A -85,B 0,C 180,E1 32429.806,E2 32429.806} C_VEL
LIN {X 0,Y 679.902,Z 1130.738,A -85,B 0,C 180,E1 32427.692,E2 32427.692} C_VEL
LIN {X 0,Y 679.907,Z 1131.822,A -85,B 0,C 180,E1 32425.711,E2 32425.711} C_VEL
LIN {X 0,Y 679.916,Z 1131.683,A -85,B 0,C 180,E1 32423.671,E2 32423.671} C_VEL
LIN {X 0,Y 679.911,Z 1129.751,A -85,B 0,C 180,E1 32421.209,E2 32421.209} C_VEL
LIN {X 0,Y 679.918,Z 1126.275,A -85,B 0,C 180,E1 32418.966,E2 32418.966} C_VEL
LIN {X 0,Y 679.936,Z 1121.028,A -85,B 0,C 180,E1 32416.664,E2 32416.664} C_VEL
LIN {X 0,Y 679.984,Z 1114.08,A -85,B 0,C 180,E1 32414.389,E2 32414.389} C_VEL
LIN {X 0,Y 680.112,Z 1106.546,A -85,B 0,C 180,E1 32412.395,E2 32412.395} C_VEL
LIN {X 0,Y 680.302,Z 1098.147,A -85,B 0,C 180,E1 32410.498,E2 32410.498} C_VEL
LIN {X 0,Y 680.563,Z 1087.177,A -85,B 0,C 180,E1 32408.364,E2 32408.364} C_VEL
LIN {X 0,Y 680.978,Z 1073.895,A -85,B 0,C 180,E1 32406.153,E2 32406.153} C_VEL
LIN {X 0,Y 681.483,Z 1060.545,A -85,B 0,C 180,E1 32404.207,E2 32404.207} C_VEL
LIN {X 0,Y 682.139,Z 1044.939,A -85,B 0,C 180,E1 32402.184,E2 32402.184} C_VEL
LIN {X 0,Y 682.962,Z 1027.251,A -85,B 0,C 180,E1 32400.168,E2 32400.168} C_VEL
LIN {X 0,Y 683.856,Z 1009.167,A -85,B 0,C 180,E1 32398.324,E2 32398.324} C_VEL
LIN {X 0,Y 685.024,Z 987.791,A -85,B 0,C 180,E1 32396.401,E2 32396.401} C_VEL
LIN {X 0,Y 686.098,Z 968.527,A -85,B 0,C 180,E1 32394.858,E2 32394.858} C_VEL
LIN {X 0,Y 687.456,Z 945.199,A -85,B 0,C 180,E1 32393.192,E2 32393.192} C_VEL
LIN {X 0,Y 688.735,Z 922.586,A -85,B 0,C 180,E1 32391.778,E2 32391.778} C_VEL
LIN {X 0,Y 689.938,Z 900.835,A -85,B 0,C 180,E1 32390.574,E2 32390.574} C_VEL
LIN {X 0,Y 691.361,Z 874.079,A -85,B 0,C 180,E1 32389.29,E2 32389.29} C_VEL
LIN {X 0,Y 692.549,Z 849.58,A -85,B 0,C 180,E1 32388.296,E2 32388.296} C_VEL
LIN {X 0,Y 693.5,Z 826.882,A -85,B 0,C 180,E1 32387.51,E2 32387.51} C_VEL
LIN {X 0,Y 694.514,Z 800.838,A -85,B 0,C 180,E1 32386.767,E2 32386.767} C_VEL
LIN {X 0,Y 695.374,Z 773.865,A -85,B 0,C 180,E1 32386.167,E2 32386.167} C_VEL
LIN {X 0,Y 695.963,Z 747.404,A -85,B 0,C 180,E1 32385.744,E2 32385.744} C_VEL
LIN {X 0,Y 698.364,Z 519.446,A -85,B 0,C 180,E1 32382.874,E2 32382.874} C_VEL
LIN {X 0,Y 699.975,Z 365.066,A -85,B 0,C 180,E1 32380.87,E2 32380.87} C_VEL
LIN {X 0,Y 689.678,Z 350.539,A -85,B 0,C 180,E1 32379.826,E2 32379.826} C_VEL
LIN {X 0,Y 686.839,Z 346.567,A -85,B 0,C 180,E1 32379.53,E2 32379.53} C_VEL
LIN {X 0,Y 684.19,Z 342.614,A -85,B 0,C 180,E1 32379.246,E2 32379.246} C_VEL
LIN {X 0,Y 681.233,Z 338.934,A -85,B 0,C 180,E1 32378.936,E2 32378.936} C_VEL
LIN {X 0,Y 680.592,Z 336.935,A -85,B 0,C 180,E1 32378.79,E2 32378.79} C_VEL
LIN {X 0,Y 680.528,Z 336.442,A -85,B 0,C 180,E1 32378.441,E2 32378.441} C_VEL
LIN {X 0,Y 680.471,Z 336.469,A -85,B 0,C 180,E1 32375.52,E2 32375.52} C_VEL
LIN {X 0,Y 680.523,Z 336.465,A -85,B 0,C 180,E1 32372.62,E2 32372.62} C_VEL
LIN {X 0,Y 680.491,Z 336.464,A -85,B 0,C 180,E1 32369.599,E2 32369.599} C_VEL
LIN {X 0,Y 680.521,Z 336.466,A -85,B 0,C 180,E1 32366.666,E2 32366.666} C_VEL
LIN {X 0,Y 680.51,Z 336.465,A -85,B 0,C 180,E1 32363.586,E2 32363.586} C_VEL
LIN {X 0,Y 680.549,Z 336.719,A -85,B 0,C 180,E1 32362.203,E2 32362.203} C_VEL
LIN {X 0,Y 682.569,Z 342.018,A -85,B 0,C 180,E1 32361.736,E2 32361.736} C_VEL
LIN {X 0,Y 688.282,Z 354.872,A -85,B 0,C 180,E1 32360.699,E2 32360.699} C_VEL
LIN {X 0,Y 697.477,Z 369.767,A -85,B 0,C 180,E1 32359.394,E2 32359.394} C_VEL
LIN {X 0,Y 698.692,Z 372.421,A -85,B 0,C 180,E1 32359.119,E2 32359.119} C_VEL
LIN {X 0,Y 696.851,Z 414.79,A -85,B 0,C 180,E1 32356.393,E2 32356.393} C_VEL
LIN {X 0,Y 696.468,Z 427.585,A -85,B 0,C 180,E1 32355.618,E2 32355.618} C_VEL
LIN {X 0,Y 700.83,Z 447.761,A -85,B 0,C 180,E1 32354.964,E2 32354.964} C_VEL
LIN {X 0,Y 698.52,Z 654.517,A -85,B 0,C 180,E1 32352.272,E2 32352.272} C_VEL
LIN {X 0,Y 696.177,Z 879.865,A -85,B 0,C 180,E1 32349.433,E2 32349.433} C_VEL
LIN {X 0,Y 695.623,Z 914.054,A -85,B 0,C 180,E1 32348.963,E2 32348.963} C_VEL
LIN {X 0,Y 694.851,Z 940.365,A -85,B 0,C 180,E1 32348.439,E2 32348.439} C_VEL
LIN {X 0,Y 693.985,Z 965.094,A -85,B 0,C 180,E1 32347.804,E2 32347.804} C_VEL
LIN {X 0,Y 692.851,Z 993.176,A -85,B 0,C 180,E1 32346.894,E2 32346.894} C_VEL
LIN {X 0,Y 691.79,Z 1015.351,A -85,B 0,C 180,E1 32346.033,E2 32346.033} C_VEL
LIN {X 0,Y 690.755,Z 1035.668,A -85,B 0,C 180,E1 32345.129,E2 32345.129} C_VEL
LIN {X 0,Y 689.673,Z 1055.669,A -85,B 0,C 180,E1 32344.122,E2 32344.122} C_VEL
LIN {X 0,Y 688.521,Z 1076.458,A -85,B 0,C 180,E1 32342.946,E2 32342.946} C_VEL
LIN {X 0,Y 687.067,Z 1101.245,A -85,B 0,C 180,E1 32341.35,E2 32341.35} C_VEL
LIN {X 0,Y 685.984,Z 1120.446,A -85,B 0,C 180,E1 32339.948,E2 32339.948} C_VEL
LIN {X 0,Y 684.982,Z 1138.821,A -85,B 0,C 180,E1 32338.463,E2 32338.463} C_VEL
LIN {X 0,Y 683.778,Z 1160.458,A -85,B 0,C 180,E1 32336.5,E2 32336.5} C_VEL
LIN {X 0,Y 682.979,Z 1176.692,A -85,B 0,C 180,E1 32334.845,E2 32334.845} C_VEL
LIN {X 0,Y 682.182,Z 1193.488,A -85,B 0,C 180,E1 32332.947,E2 32332.947} C_VEL
LIN {X 0,Y 681.485,Z 1209.918,A -85,B 0,C 180,E1 32330.832,E2 32330.832} C_VEL
LIN {X 0,Y 681.038,Z 1222.57,A -85,B 0,C 180,E1 32329,E2 32329} C_VEL
LIN {X 0,Y 680.647,Z 1234.892,A -85,B 0,C 180,E1 32326.993,E2 32326.993} C_VEL
LIN {X 0,Y 680.343,Z 1246.839,A -85,B 0,C 180,E1 32324.729,E2 32324.729} C_VEL
LIN {X 0,Y 680.158,Z 1255.795,A -85,B 0,C 180,E1 32322.739,E2 32322.739} C_VEL
LIN {X 0,Y 680.022,Z 1262.745,A -85,B 0,C 180,E1 32320.934,E2 32320.934} C_VEL
LIN {X 0,Y 679.93,Z 1268.309,A -85,B 0,C 180,E1 32319.224,E2 32319.224} C_VEL
LIN {X 0,Y 679.926,Z 1273.37,A -85,B 0,C 180,E1 32317.35,E2 32317.35} C_VEL
LIN {X 0,Y 679.918,Z 1277.928,A -85,B 0,C 180,E1 32315.062,E2 32315.062} C_VEL
